KUKA KRL program: EPS_2_251692_SAMH06_A_20251205090702.src

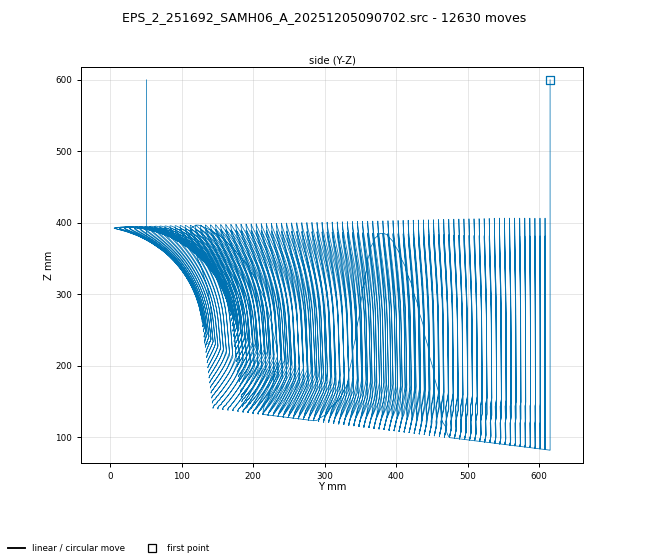
[picture p0: tool path of EPS_2_251692_SAMH06_A_20251205090702.src, 12630 of 12632 moves have a stored position in this frame; points joined in program order, loops and branches not executed]
&ACCESS RVP
&REL 4
&COMMENT QRS 19112012
&PARAM EDITMASK = *
DEF PART()
EXT BAS (BAS_COMMAND :IN,REAL :IN )
INT I
BAS (#INITMOV,0 )

;KUKA QRS Post kuka4.cps  Date:22-06-2017 !

File_ID=2948

QRS_PRE_INIT()

;Init var - Until changes are made in qrs_pre_init
Outlet_Square_prg=0
Inlet_1_Square_prg=0
Inlet_2_Square_prg=0
Inlet_3_Square_prg=0
Inlet_4_Square_prg=0
Inlet_5_Square_prg=0

Outlet_1={X 0.000, Y 543.810, Z 281.000, B 0.000, E1 0.000 }
Inlet_1={X 0.000, Y 545.610, Z 256.000, B 0.000, E1 186.000 }
Outlet_1_type=251
Inlet_1_type=251
;QRS#1=Sidecore dimensions
;QRS#2=250-10" PVC SDR 35
;QRS#3=250-10" PVC SDR 35
;QRS#4=
;QRS#5=
;QRS#6=
;QRS#7=
;QRS#8=
;QRS#9=14M PSX
;QRS#10=14M PSX
;QRS#11=
;QRS#12=
;QRS#13=
;QRS#14=
;QRS#15=
;QRS#16=1220x127x686 2,25'
;QRS#17=EPS Height
;QRS#18=406,5
;QRS#19=*
;QRS#20= UPDATED VERSION 22-06-2017
;QRS#21=*
Outlet_Square=0100
Inlet_1_Square=0100
Inlet_2_Square=0
Inlet_3_Square=0
Inlet_4_Square=0
Inlet_5_Square=0
Mill_Square=1
Outlet_Square_Prg=205
Inlet_1_Square_prg=205

QRS_INIT()

$ADVANCE=5

; T1
PTP {E1 173.621,E2 173.621}
PTP {X 0,Y 615.479,A -85,B 0,C 180,E1 173.621,E2 173.621,E3 0,E4 0,E5 0,E6 0}
QRS_SPEED_INIT()
LIN {X 0,Y 615.479,Z 600,A -85,B 0,C 180,E1 173.621,E2 173.621,E3 0,E4 0,E5 0,E6 0} C_VEL
LIN {X 0,Y 615.479,Z 91.999,A -85,B 0,C 180,E1 173.621,E2 173.621} C_VEL
LIN {X 0,Y 615.479,Z 83.818,A -85,B 0,C 180,E1 173.621,E2 173.621} C_VEL
LIN {X 0,Y 615.469,Z 81.818,A -85,B 0,C 180,E1 173.435,E2 173.435} C_VEL
LIN {X 0,Y 615.495,Z 81.807,A -85,B 0,C 180,E1 170.801,E2 170.801} C_VEL
LIN {X 0,Y 615.489,Z 81.826,A -85,B 0,C 180,E1 168.139,E2 168.139} C_VEL
LIN {X 0,Y 615.464,Z 81.815,A -85,B 0,C 180,E1 165.45,E2 165.45} C_VEL
LIN {X 0,Y 615.485,Z 81.814,A -85,B 0,C 180,E1 162.729,E2 162.729} C_VEL
LIN {X 0,Y 615.469,Z 81.82,A -85,B 0,C 180,E1 159.966,E2 159.966} C_VEL
LIN {X 0,Y 615.486,Z 81.81,A -85,B 0,C 180,E1 157.155,E2 157.155} C_VEL
LIN {X 0,Y 615.476,Z 81.822,A -85,B 0,C 180,E1 154.284,E2 154.284} C_VEL
LIN {X 0,Y 615.47,Z 81.812,A -85,B 0,C 180,E1 151.552,E2 151.552} C_VEL
LIN {X 0,Y 615.492,Z 81.82,A -85,B 0,C 180,E1 148.913,E2 148.913} C_VEL
LIN {X 0,Y 615.47,Z 81.821,A -85,B 0,C 180,E1 146.468,E2 146.468} C_VEL
LIN {X 0,Y 615.458,Z 81.816,A -85,B 0,C 180,E1 144.17,E2 144.17} C_VEL
LIN {X 0,Y 615.467,Z 81.813,A -85,B 0,C 180,E1 141.93,E2 141.93} C_VEL
LIN {X 0,Y 615.492,Z 81.815,A -85,B 0,C 180,E1 139.394,E2 139.394} C_VEL
LIN {X 0,Y 615.466,Z 81.821,A -85,B 0,C 180,E1 136.753,E2 136.753} C_VEL
LIN {X 0,Y 615.474,Z 81.812,A -85,B 0,C 180,E1 133.996,E2 133.996} C_VEL
LIN {X 0,Y 615.475,Z 81.823,A -85,B 0,C 180,E1 131.093,E2 131.093} C_VEL
LIN {X 0,Y 615.459,Z 81.82,A -85,B 0,C 180,E1 128.906,E2 128.906} C_VEL
LIN {X 0,Y 615.46,Z 81.814,A -85,B 0,C 180,E1 126.426,E2 126.426} C_VEL
LIN {X 0,Y 615.494,Z 81.826,A -85,B 0,C 180,E1 123.535,E2 123.535} C_VEL
LIN {X 0,Y 615.45,Z 81.818,A -85,B 0,C 180,E1 120.922,E2 120.922} C_VEL
LIN {X 0,Y 615.474,Z 81.813,A -85,B 0,C 180,E1 118.447,E2 118.447} C_VEL
LIN {X 0,Y 615.471,Z 81.823,A -85,B 0,C 180,E1 115.565,E2 115.565} C_VEL
LIN {X 0,Y 615.465,Z 81.822,A -85,B 0,C 180,E1 113.557,E2 113.557} C_VEL
LIN {X 0,Y 615.453,Z 81.82,A -85,B 0,C 180,E1 111.433,E2 111.433} C_VEL
LIN {X 0,Y 615.447,Z 81.819,A -85,B 0,C 180,E1 109.339,E2 109.339} C_VEL
LIN {X 0,Y 615.485,Z 81.814,A -85,B 0,C 180,E1 106.587,E2 106.587} C_VEL
LIN {X 0,Y 615.468,Z 81.896,A -85,B 0,C 180,E1 104.866,E2 104.866} C_VEL
LIN {X 0,Y 615.446,Z 101.823,A -85,B 0,C 180,E1 102.029,E2 102.029} C_VEL
LIN {X 0,Y 615.452,Z 119.452,A -85,B 0,C 180,E1 99.551,E2 99.551} C_VEL
LIN {X 0,Y 615.46,Z 256.695,A -85,B 0,C 180,E1 97.896,E2 97.896} C_VEL
LIN {X 0,Y 615.48,Z 271.017,A -85,B 0,C 180,E1 97.587,E2 97.587} C_VEL
LIN {X 0,Y 615.491,Z 285.222,A -85,B 0,C 180,E1 97.136,E2 97.136} C_VEL
LIN {X 0,Y 615.494,Z 298.839,A -85,B 0,C 180,E1 96.556,E2 96.556} C_VEL
LIN {X 0,Y 615.49,Z 311.023,A -85,B 0,C 180,E1 95.898,E2 95.898} C_VEL
LIN {X 0,Y 615.498,Z 322.188,A -85,B 0,C 180,E1 95.159,E2 95.159} C_VEL
LIN {X 0,Y 615.497,Z 333.436,A -85,B 0,C 180,E1 94.256,E2 94.256} C_VEL
LIN {X 0,Y 615.496,Z 343.522,A -85,B 0,C 180,E1 93.273,E2 93.273} C_VEL
LIN {X 0,Y 615.497,Z 351.879,A -85,B 0,C 180,E1 92.29,E2 92.29} C_VEL
LIN {X 0,Y 615.496,Z 359.883,A -85,B 0,C 180,E1 91.145,E2 91.145} C_VEL
LIN {X 0,Y 615.494,Z 366.357,A -85,B 0,C 180,E1 90,E2 90} C_VEL
LIN {X 0,Y 615.498,Z 372.115,A -85,B 0,C 180,E1 88.691,E2 88.691} C_VEL
LIN {X 0,Y 615.493,Z 376.34,A -85,B 0,C 180,E1 87.382,E2 87.382} C_VEL
LIN {X 0,Y 615.493,Z 379.15,A -85,B 0,C 180,E1 86.071,E2 86.071} C_VEL
LIN {X 0,Y 615.49,Z 380.617,A -85,B 0,C 180,E1 84.759,E2 84.759} C_VEL
LIN {X 0,Y 615.496,Z 380.768,A -85,B 0,C 180,E1 83.418,E2 83.418} C_VEL
LIN {X 0,Y 615.493,Z 379.611,A -85,B 0,C 180,E1 82.124,E2 82.124} C_VEL
LIN {X 0,Y 615.496,Z 377.073,A -85,B 0,C 180,E1 80.801,E2 80.801} C_VEL
LIN {X 0,Y 615.494,Z 373.067,A -85,B 0,C 180,E1 79.473,E2 79.473} C_VEL
LIN {X 0,Y 615.494,Z 367.474,A -85,B 0,C 180,E1 78.139,E2 78.139} C_VEL
LIN {X 0,Y 615.494,Z 361.111,A -85,B 0,C 180,E1 76.967,E2 76.967} C_VEL
LIN {X 0,Y 615.495,Z 352.912,A -85,B 0,C 180,E1 75.758,E2 75.758} C_VEL
LIN {X 0,Y 615.495,Z 344.746,A -85,B 0,C 180,E1 74.774,E2 74.774} C_VEL
LIN {X 0,Y 615.498,Z 335.393,A -85,B 0,C 180,E1 73.832,E2 73.832} C_VEL
LIN {X 0,Y 615.497,Z 324.257,A -85,B 0,C 180,E1 72.901,E2 72.901} C_VEL
LIN {X 0,Y 615.495,Z 313,A -85,B 0,C 180,E1 72.129,E2 72.129} C_VEL
LIN {X 0,Y 615.497,Z 301.366,A -85,B 0,C 180,E1 71.475,E2 71.475} C_VEL
LIN {X 0,Y 615.483,Z 288.017,A -85,B 0,C 180,E1 70.878,E2 70.878} C_VEL
LIN {X 0,Y 615.495,Z 275.413,A -85,B 0,C 180,E1 70.445,E2 70.445} C_VEL
LIN {X 0,Y 615.477,Z 261.216,A -85,B 0,C 180,E1 70.097,E2 70.097} C_VEL
LIN {X 0,Y 615.478,Z 244.533,A -85,B 0,C 180,E1 69.852,E2 69.852} C_VEL
LIN {X 0,Y 615.468,Z 119.526,A -85,B 0,C 180,E1 68.37,E2 68.37} C_VEL
LIN {X 0,Y 615.494,Z 99.456,A -85,B 0,C 180,E1 65.549,E2 65.549} C_VEL
LIN {X 0,Y 615.42,Z 81.825,A -85,B 0,C 180,E1 63.023,E2 63.023} C_VEL
LIN {X 0,Y 615.417,Z 81.825,A -85,B 0,C 180,E1 60.59,E2 60.59} C_VEL
LIN {X 0,Y 615.445,Z 81.825,A -85,B 0,C 180,E1 58.312,E2 58.312} C_VEL
LIN {X 0,Y 615.494,Z 81.826,A -85,B 0,C 180,E1 55.978,E2 55.978} C_VEL
LIN {X 0,Y 615.443,Z 81.823,A -85,B 0,C 180,E1 53.572,E2 53.572} C_VEL
LIN {X 0,Y 615.424,Z 81.824,A -85,B 0,C 180,E1 50.946,E2 50.946} C_VEL
LIN {X 0,Y 615.464,Z 81.825,A -85,B 0,C 180,E1 48.524,E2 48.524} C_VEL
LIN {X 0,Y 615.449,Z 81.822,A -85,B 0,C 180,E1 45.847,E2 45.847} C_VEL
LIN {X 0,Y 615.428,Z 81.823,A -85,B 0,C 180,E1 43.25,E2 43.25} C_VEL
LIN {X 0,Y 615.487,Z 81.826,A -85,B 0,C 180,E1 40.607,E2 40.607} C_VEL
LIN {X 0,Y 615.449,Z 81.819,A -85,B 0,C 180,E1 38.007,E2 38.007} C_VEL
LIN {X 0,Y 615.432,Z 81.821,A -85,B 0,C 180,E1 35.62,E2 35.62} C_VEL
LIN {X 0,Y 615.453,Z 81.823,A -85,B 0,C 180,E1 33.239,E2 33.239} C_VEL
LIN {X 0,Y 615.49,Z 81.827,A -85,B 0,C 180,E1 30.92,E2 30.92} C_VEL
LIN {X 0,Y 615.437,Z 81.82,A -85,B 0,C 180,E1 27.918,E2 27.918} C_VEL
LIN {X 0,Y 615.452,Z 81.822,A -85,B 0,C 180,E1 25.562,E2 25.562} C_VEL
LIN {X 0,Y 615.486,Z 81.816,A -85,B 0,C 180,E1 22.845,E2 22.845} C_VEL
LIN {X 0,Y 615.443,Z 81.82,A -85,B 0,C 180,E1 20.034,E2 20.034} C_VEL
LIN {X 0,Y 615.496,Z 81.821,A -85,B 0,C 180,E1 17.27,E2 17.27} C_VEL
LIN {X 0,Y 615.448,Z 81.817,A -85,B 0,C 180,E1 14.55,E2 14.55} C_VEL
LIN {X 0,Y 615.449,Z 81.817,A -85,B 0,C 180,E1 12.531,E2 12.531} C_VEL
LIN {X 0,Y 615.48,Z 81.824,A -85,B 0,C 180,E1 9.862,E2 9.862} C_VEL
LIN {X 0,Y 615.481,Z 81.813,A -85,B 0,C 180,E1 7.216,E2 7.216} C_VEL
LIN {X 0,Y 615.452,Z 81.818,A -85,B 0,C 180,E1 4.585,E2 4.585} C_VEL
LIN {X 0,Y 615.498,Z 81.825,A -85,B 0,C 180,E1 1.963,E2 1.963} C_VEL
LIN {X 0,Y 615.476,Z 81.812,A -85,B 0,C 180,E1 -0.654,E2 -0.654} C_VEL
LIN {X 0,Y 615.459,Z 81.819,A -85,B 0,C 180,E1 -3.273,E2 -3.273} C_VEL
LIN {X 0,Y 615.493,Z 81.82,A -85,B 0,C 180,E1 -5.898,E2 -5.898} C_VEL
LIN {X 0,Y 615.474,Z 81.811,A -85,B 0,C 180,E1 -8.537,E2 -8.537} C_VEL
LIN {X 0,Y 615.47,Z 81.821,A -85,B 0,C 180,E1 -11.193,E2 -11.193} C_VEL
LIN {X 0,Y 615.49,Z 81.813,A -85,B 0,C 180,E1 -13.933,E2 -13.933} C_VEL
LIN {X 0,Y 615.462,Z 81.815,A -85,B 0,C 180,E1 -16.587,E2 -16.587} C_VEL
LIN {X 0,Y 615.493,Z 81.823,A -85,B 0,C 180,E1 -19.338,E2 -19.338} C_VEL
LIN {X 0,Y 615.469,Z 81.813,A -85,B 0,C 180,E1 -22.342,E2 -22.342} C_VEL
LIN {X 0,Y 615.492,Z 81.826,A -85,B 0,C 180,E1 -24.992,E2 -24.992} C_VEL
LIN {X 0,Y 615.484,Z 81.809,A -85,B 0,C 180,E1 -27.915,E2 -27.915} C_VEL
LIN {X 0,Y 615.471,Z 81.814,A -85,B 0,C 180,E1 -30.161,E2 -30.161} C_VEL
LIN {X 0,Y 615.478,Z 81.82,A -85,B 0,C 180,E1 -32.458,E2 -32.458} C_VEL
LIN {X 0,Y 615.49,Z 81.822,A -85,B 0,C 180,E1 -34.815,E2 -34.815} C_VEL
LIN {X 0,Y 615.487,Z 81.81,A -85,B 0,C 180,E1 -37.242,E2 -37.242} C_VEL
LIN {X 0,Y 615.476,Z 81.818,A -85,B 0,C 180,E1 -40.088,E2 -40.088} C_VEL
LIN {X 0,Y 615.497,Z 81.825,A -85,B 0,C 180,E1 -42.352,E2 -42.352} C_VEL
LIN {X 0,Y 615.481,Z 81.811,A -85,B 0,C 180,E1 -45.069,E2 -45.069} C_VEL
LIN {X 0,Y 615.483,Z 81.82,A -85,B 0,C 180,E1 -47.92,E2 -47.92} C_VEL
LIN {X 0,Y 615.486,Z 81.823,A -85,B 0,C 180,E1 -50.25,E2 -50.25} C_VEL
LIN {X 0,Y 615.489,Z 81.808,A -85,B 0,C 180,E1 -53.063,E2 -53.063} C_VEL
LIN {X 0,Y 615.492,Z 81.823,A -85,B 0,C 180,E1 -55.978,E2 -55.978} C_VEL
LIN {X 0,Y 615.488,Z 81.809,A -85,B 0,C 180,E1 -58.914,E2 -58.914} C_VEL
LIN {X 0,Y 615.492,Z 81.822,A -85,B 0,C 180,E1 -61.549,E2 -61.549} C_VEL
LIN {X 0,Y 615.479,Z 81.81,A -85,B 0,C 180,E1 -64.433,E2 -64.433} C_VEL
LIN {X 0,Y 615.492,Z 81.815,A -85,B 0,C 180,E1 -66.711,E2 -66.711} C_VEL
LIN {X 0,Y 615.483,Z 104.503,A -85,B 0,C 180,E1 -69.576,E2 -69.576} C_VEL
LIN {X 0,Y 615.496,Z 127.142,A -85,B 0,C 180,E1 -72.387,E2 -72.387} C_VEL
LIN {X 0,Y 615.494,Z 143.505,A -85,B 0,C 180,E1 -74.392,E2 -74.392} C_VEL
LIN {X 0,Y 615.478,Z 281.308,A -85,B 0,C 180,E1 -76.052,E2 -76.052} C_VEL
LIN {X 0,Y 615.489,Z 294.854,A -85,B 0,C 180,E1 -76.336,E2 -76.336} C_VEL
LIN {X 0,Y 615.488,Z 308.565,A -85,B 0,C 180,E1 -76.757,E2 -76.757} C_VEL
LIN {X 0,Y 615.494,Z 321.835,A -85,B 0,C 180,E1 -77.302,E2 -77.302} C_VEL
LIN {X 0,Y 615.483,Z 334.599,A -85,B 0,C 180,E1 -77.972,E2 -77.972} C_VEL
LIN {X 0,Y 615.499,Z 347.339,A -85,B 0,C 180,E1 -78.807,E2 -78.807} C_VEL
LIN {X 0,Y 615.498,Z 357.747,A -85,B 0,C 180,E1 -79.639,E2 -79.639} C_VEL
LIN {X 0,Y 615.496,Z 368.087,A -85,B 0,C 180,E1 -80.636,E2 -80.636} C_VEL
LIN {X 0,Y 615.497,Z 376.602,A -85,B 0,C 180,E1 -81.629,E2 -81.629} C_VEL
LIN {X 0,Y 615.496,Z 384.726,A -85,B 0,C 180,E1 -82.784,E2 -82.784} C_VEL
LIN {X 0,Y 615.496,Z 390.429,A -85,B 0,C 180,E1 -83.772,E2 -83.772} C_VEL
LIN {X 0,Y 615.495,Z 395.08,A -85,B 0,C 180,E1 -84.759,E2 -84.759} C_VEL
LIN {X 0,Y 615.496,Z 399.901,A -85,B 0,C 180,E1 -86.071,E2 -86.071} C_VEL
LIN {X 0,Y 615.495,Z 403.252,A -85,B 0,C 180,E1 -87.382,E2 -87.382} C_VEL
LIN {X 0,Y 615.49,Z 405.228,A -85,B 0,C 180,E1 -88.691,E2 -88.691} C_VEL
LIN {X 0,Y 615.493,Z 405.889,A -85,B 0,C 180,E1 -90,E2 -90} C_VEL
LIN {X 0,Y 615.49,Z 405.229,A -85,B 0,C 180,E1 -91.308,E2 -91.308} C_VEL
LIN {X 0,Y 615.495,Z 403.252,A -85,B 0,C 180,E1 -92.618,E2 -92.618} C_VEL
LIN {X 0,Y 615.496,Z 399.901,A -85,B 0,C 180,E1 -93.928,E2 -93.928} C_VEL
LIN {X 0,Y 615.495,Z 395.081,A -85,B 0,C 180,E1 -95.241,E2 -95.241} C_VEL
LIN {X 0,Y 615.495,Z 388.629,A -85,B 0,C 180,E1 -96.556,E2 -96.556} C_VEL
LIN {X 0,Y 615.498,Z 381.441,A -85,B 0,C 180,E1 -97.71,E2 -97.71} C_VEL
LIN {X 0,Y 615.497,Z 373.904,A -85,B 0,C 180,E1 -98.702,E2 -98.702} C_VEL
LIN {X 0,Y 615.496,Z 364.854,A -85,B 0,C 180,E1 -99.696,E2 -99.696} C_VEL
LIN {X 0,Y 615.497,Z 354.758,A -85,B 0,C 180,E1 -100.618,E2 -100.618} C_VEL
LIN {X 0,Y 615.498,Z 343.859,A -85,B 0,C 180,E1 -101.443,E2 -101.443} C_VEL
LIN {X 0,Y 615.484,Z 331.708,A -85,B 0,C 180,E1 -102.195,E2 -102.195} C_VEL
LIN {X 0,Y 615.486,Z 318.093,A -85,B 0,C 180,E1 -102.865,E2 -102.865} C_VEL
LIN {X 0,Y 615.488,Z 304.838,A -85,B 0,C 180,E1 -103.369,E2 -103.369} C_VEL
LIN {X 0,Y 615.487,Z 291.29,A -85,B 0,C 180,E1 -103.748,E2 -103.748} C_VEL
LIN {X 0,Y 615.479,Z 277.161,A -85,B 0,C 180,E1 -104.007,E2 -104.007} C_VEL
LIN {X 0,Y 615.494,Z 143.507,A -85,B 0,C 180,E1 -105.607,E2 -105.607} C_VEL
LIN {X 0,Y 615.471,Z 120.463,A -85,B 0,C 180,E1 -108.439,E2 -108.439} C_VEL
LIN {X 0,Y 615.472,Z 99.26,A -85,B 0,C 180,E1 -111.081,E2 -111.081} C_VEL
LIN {X 0,Y 615.494,Z 81.808,A -85,B 0,C 180,E1 -113.311,E2 -113.311} C_VEL
LIN {X 0,Y 615.473,Z 81.813,A -85,B 0,C 180,E1 -115.716,E2 -115.716} C_VEL
LIN {X 0,Y 615.493,Z 81.823,A -85,B 0,C 180,E1 -118.451,E2 -118.451} C_VEL
LIN {X 0,Y 615.486,Z 81.809,A -85,B 0,C 180,E1 -121.086,E2 -121.086} C_VEL
LIN {X 0,Y 615.474,Z 81.814,A -85,B 0,C 180,E1 -123.532,E2 -123.532} C_VEL
LIN {X 0,Y 615.481,Z 81.82,A -85,B 0,C 180,E1 -125.833,E2 -125.833} C_VEL
LIN {X 0,Y 615.488,Z 81.826,A -85,B 0,C 180,E1 -128.068,E2 -128.068} C_VEL
LIN {X 0,Y 615.479,Z 81.812,A -85,B 0,C 180,E1 -130.607,E2 -130.607} C_VEL
LIN {X 0,Y 615.474,Z 81.814,A -85,B 0,C 180,E1 -133.246,E2 -133.246} C_VEL
LIN {X 0,Y 615.485,Z 81.82,A -85,B 0,C 180,E1 -136.003,E2 -136.003} C_VEL
LIN {X 0,Y 615.487,Z 81.809,A -85,B 0,C 180,E1 -138.526,E2 -138.526} C_VEL
LIN {X 0,Y 615.477,Z 81.815,A -85,B 0,C 180,E1 -141.095,E2 -141.095} C_VEL
LIN {X 0,Y 615.483,Z 81.827,A -85,B 0,C 180,E1 -143.575,E2 -143.575} C_VEL
LIN {X 0,Y 615.494,Z 81.807,A -85,B 0,C 180,E1 -146.464,E2 -146.464} C_VEL
LIN {X 0,Y 615.484,Z 81.82,A -85,B 0,C 180,E1 -149.08,E2 -149.08} C_VEL
LIN {X 0,Y 615.477,Z 81.82,A -85,B 0,C 180,E1 -151.551,E2 -151.551} C_VEL
LIN {X 0,Y 615.486,Z 81.81,A -85,B 0,C 180,E1 -154.431,E2 -154.431} C_VEL
LIN {X 0,Y 615.485,Z 81.825,A -85,B 0,C 180,E1 -157.155,E2 -157.155} C_VEL
LIN {X 0,Y 615.485,Z 81.809,A -85,B 0,C 180,E1 -159.967,E2 -159.967} C_VEL
LIN {X 0,Y 615.488,Z 81.822,A -85,B 0,C 180,E1 -162.73,E2 -162.73} C_VEL
LIN {X 0,Y 615.474,Z 81.813,A -85,B 0,C 180,E1 -165.451,E2 -165.451} C_VEL
LIN {X 0,Y 615.485,Z 81.813,A -85,B 0,C 180,E1 -168.139,E2 -168.139} C_VEL
LIN {X 0,Y 615.484,Z 81.822,A -85,B 0,C 180,E1 -170.801,E2 -170.801} C_VEL
LIN {X 0,Y 615.481,Z 81.81,A -85,B 0,C 180,E1 -173.443,E2 -173.443} C_VEL
LIN {X 0,Y 615.485,Z 81.817,A -85,B 0,C 180,E1 -176.072,E2 -176.072} C_VEL
LIN {X 0,Y 615.475,Z 81.82,A -85,B 0,C 180,E1 -178.691,E2 -178.691} C_VEL
LIN {X 0,Y 615.486,Z 81.808,A -85,B 0,C 180,E1 -181.309,E2 -181.309} C_VEL
LIN {X 0,Y 615.488,Z 81.819,A -85,B 0,C 180,E1 -183.929,E2 -183.929} C_VEL
LIN {X 0,Y 615.469,Z 81.818,A -85,B 0,C 180,E1 -186.565,E2 -186.565} C_VEL
LIN {X 0,Y 614.805,Z 81.958,A -85,B 0,C 180,E1 -187.111,E2 -187.111} C_VEL
LIN {X 0,Y 611.984,Z 82.383,A -85,B 0,C 180,E1 -187.997,E2 -187.997} C_VEL
LIN {X 0,Y 609.596,Z 82.686,A -85,B 0,C 180,E1 -188.71,E2 -188.71} C_VEL
LIN {X 0,Y 608.558,Z 82.802,A -85,B 0,C 180,E1 -189.259,E2 -189.259} C_VEL
LIN {X 0,Y 608.467,Z 82.813,A -85,B 0,C 180,E1 -189.445,E2 -189.445} C_VEL
LIN {X 0,Y 608.46,Z 82.821,A -85,B 0,C 180,E1 -192,E2 -192} C_VEL
LIN {X 0,Y 608.463,Z 82.812,A -85,B 0,C 180,E1 -194.721,E2 -194.721} C_VEL
LIN {X 0,Y 608.45,Z 82.819,A -85,B 0,C 180,E1 -197.477,E2 -197.477} C_VEL
LIN {X 0,Y 608.447,Z 82.815,A -85,B 0,C 180,E1 -200.275,E2 -200.275} C_VEL
LIN {X 0,Y 608.458,Z 82.812,A -85,B 0,C 180,E1 -202.477,E2 -202.477} C_VEL
LIN {X 0,Y 608.454,Z 82.82,A -85,B 0,C 180,E1 -205.301,E2 -205.301} C_VEL
LIN {X 0,Y 608.442,Z 82.822,A -85,B 0,C 180,E1 -207.519,E2 -207.519} C_VEL
LIN {X 0,Y 608.445,Z 82.815,A -85,B 0,C 180,E1 -209.968,E2 -209.968} C_VEL
LIN {X 0,Y 608.455,Z 82.817,A -85,B 0,C 180,E1 -212.88,E2 -212.88} C_VEL
LIN {X 0,Y 608.432,Z 82.823,A -85,B 0,C 180,E1 -215.279,E2 -215.279} C_VEL
LIN {X 0,Y 608.455,Z 82.813,A -85,B 0,C 180,E1 -217.748,E2 -217.748} C_VEL
LIN {X 0,Y 608.445,Z 82.815,A -85,B 0,C 180,E1 -220.329,E2 -220.329} C_VEL
LIN {X 0,Y 608.451,Z 82.822,A -85,B 0,C 180,E1 -222.96,E2 -222.96} C_VEL
LIN {X 0,Y 608.436,Z 82.815,A -85,B 0,C 180,E1 -225.738,E2 -225.738} C_VEL
LIN {X 0,Y 608.454,Z 82.813,A -85,B 0,C 180,E1 -227.938,E2 -227.938} C_VEL
LIN {X 0,Y 608.439,Z 82.824,A -85,B 0,C 180,E1 -230.707,E2 -230.707} C_VEL
LIN {X 0,Y 608.428,Z 82.818,A -85,B 0,C 180,E1 -233.083,E2 -233.083} C_VEL
LIN {X 0,Y 608.452,Z 82.813,A -85,B 0,C 180,E1 -235.53,E2 -235.53} C_VEL
LIN {X 0,Y 608.462,Z 82.814,A -85,B 0,C 180,E1 -237.906,E2 -237.906} C_VEL
LIN {X 0,Y 608.479,Z 82.818,A -85,B 0,C 180,E1 -240.221,E2 -240.221} C_VEL
LIN {X 0,Y 608.429,Z 82.818,A -85,B 0,C 180,E1 -242.803,E2 -242.803} C_VEL
LIN {X 0,Y 608.443,Z 82.815,A -85,B 0,C 180,E1 -245.429,E2 -245.429} C_VEL
LIN {X 0,Y 608.453,Z 82.819,A -85,B 0,C 180,E1 -248.308,E2 -248.308} C_VEL
LIN {X 0,Y 608.447,Z 82.814,A -85,B 0,C 180,E1 -251.13,E2 -251.13} C_VEL
LIN {X 0,Y 608.454,Z 82.823,A -85,B 0,C 180,E1 -253.906,E2 -253.906} C_VEL
LIN {X 0,Y 608.443,Z 82.879,A -85,B 0,C 180,E1 -255.022,E2 -255.022} C_VEL
LIN {X 0,Y 608.505,Z 100.007,A -85,B 0,C 180,E1 -257.493,E2 -257.493} C_VEL
LIN {X 0,Y 608.468,Z 119.013,A -85,B 0,C 180,E1 -260.191,E2 -260.191} C_VEL
LIN {X 0,Y 608.509,Z 119.95,A -85,B 0,C 180,E1 -260.286,E2 -260.286} C_VEL
LIN {X 0,Y 608.592,Z 255.971,A -85,B 0,C 180,E1 -261.93,E2 -261.93} C_VEL
LIN {X 0,Y 608.571,Z 270.582,A -85,B 0,C 180,E1 -262.243,E2 -262.243} C_VEL
LIN {X 0,Y 608.587,Z 283.896,A -85,B 0,C 180,E1 -262.661,E2 -262.661} C_VEL
LIN {X 0,Y 608.544,Z 297.268,A -85,B 0,C 180,E1 -263.219,E2 -263.219} C_VEL
LIN {X 0,Y 608.526,Z 309.517,A -85,B 0,C 180,E1 -263.867,E2 -263.867} C_VEL
LIN {X 0,Y 608.502,Z 322.152,A -85,B 0,C 180,E1 -264.699,E2 -264.699} C_VEL
LIN {X 0,Y 608.49,Z 332.525,A -85,B 0,C 180,E1 -265.529,E2 -265.529} C_VEL
LIN {X 0,Y 608.472,Z 342.87,A -85,B 0,C 180,E1 -266.524,E2 -266.524} C_VEL
LIN {X 0,Y 608.464,Z 351.439,A -85,B 0,C 180,E1 -267.518,E2 -267.518} C_VEL
LIN {X 0,Y 608.45,Z 359.687,A -85,B 0,C 180,E1 -268.676,E2 -268.676} C_VEL
LIN {X 0,Y 608.441,Z 365.452,A -85,B 0,C 180,E1 -269.669,E2 -269.669} C_VEL
LIN {X 0,Y 608.448,Z 371.636,A -85,B 0,C 180,E1 -270.993,E2 -270.993} C_VEL
LIN {X 0,Y 608.441,Z 375.17,A -85,B 0,C 180,E1 -271.986,E2 -271.986} C_VEL
LIN {X 0,Y 608.418,Z 378.646,A -85,B 0,C 180,E1 -273.311,E2 -273.311} C_VEL
LIN {X 0,Y 608.429,Z 380.732,A -85,B 0,C 180,E1 -274.638,E2 -274.638} C_VEL
LIN {X 0,Y 608.431,Z 381.488,A -85,B 0,C 180,E1 -275.967,E2 -275.967} C_VEL
LIN {X 0,Y 608.42,Z 380.907,A -85,B 0,C 180,E1 -277.3,E2 -277.3} C_VEL
LIN {X 0,Y 608.42,Z 378.953,A -85,B 0,C 180,E1 -278.637,E2 -278.637} C_VEL
LIN {X 0,Y 608.434,Z 375.573,A -85,B 0,C 180,E1 -279.978,E2 -279.978} C_VEL
LIN {X 0,Y 608.429,Z 370.663,A -85,B 0,C 180,E1 -281.325,E2 -281.325} C_VEL
LIN {X 0,Y 608.457,Z 365.899,A -85,B 0,C 180,E1 -282.338,E2 -282.338} C_VEL
LIN {X 0,Y 608.459,Z 358.935,A -85,B 0,C 180,E1 -283.527,E2 -283.527} C_VEL
LIN {X 0,Y 608.457,Z 351.621,A -85,B 0,C 180,E1 -284.55,E2 -284.55} C_VEL
LIN {X 0,Y 608.471,Z 342.76,A -85,B 0,C 180,E1 -285.578,E2 -285.578} C_VEL
LIN {X 0,Y 608.495,Z 332.04,A -85,B 0,C 180,E1 -286.603,E2 -286.603} C_VEL
LIN {X 0,Y 608.511,Z 321.001,A -85,B 0,C 180,E1 -287.475,E2 -287.475} C_VEL
LIN {X 0,Y 608.524,Z 309.03,A -85,B 0,C 180,E1 -288.252,E2 -288.252} C_VEL
LIN {X 0,Y 608.543,Z 297.362,A -85,B 0,C 180,E1 -288.867,E2 -288.867} C_VEL
LIN {X 0,Y 608.577,Z 283.761,A -85,B 0,C 180,E1 -289.435,E2 -289.435} C_VEL
LIN {X 0,Y 608.58,Z 269.596,A -85,B 0,C 180,E1 -289.874,E2 -289.874} C_VEL
LIN {X 0,Y 608.608,Z 255.992,A -85,B 0,C 180,E1 -290.159,E2 -290.159} C_VEL
LIN {X 0,Y 608.555,Z 120.203,A -85,B 0,C 180,E1 -291.8,E2 -291.8} C_VEL
LIN {X 0,Y 608.471,Z 119.536,A -85,B 0,C 180,E1 -291.825,E2 -291.825} C_VEL
LIN {X 0,Y 608.52,Z 100.202,A -85,B 0,C 180,E1 -294.568,E2 -294.568} C_VEL
LIN {X 0,Y 608.494,Z 83.884,A -85,B 0,C 180,E1 -296.92,E2 -296.92} C_VEL
LIN {X 0,Y 608.4,Z 82.821,A -85,B 0,C 180,E1 -297.12,E2 -297.12} C_VEL
LIN {X 0,Y 608.448,Z 82.821,A -85,B 0,C 180,E1 -299.968,E2 -299.968} C_VEL
LIN {X 0,Y 608.413,Z 82.818,A -85,B 0,C 180,E1 -302.882,E2 -302.882} C_VEL
LIN {X 0,Y 608.404,Z 82.82,A -85,B 0,C 180,E1 -305.28,E2 -305.28} C_VEL
LIN {X 0,Y 608.422,Z 82.821,A -85,B 0,C 180,E1 -308.234,E2 -308.234} C_VEL
LIN {X 0,Y 608.435,Z 82.817,A -85,B 0,C 180,E1 -310.327,E2 -310.327} C_VEL
LIN {X 0,Y 608.398,Z 82.821,A -85,B 0,C 180,E1 -312.965,E2 -312.965} C_VEL
LIN {X 0,Y 608.448,Z 82.821,A -85,B 0,C 180,E1 -315.737,E2 -315.737} C_VEL
LIN {X 0,Y 608.445,Z 82.817,A -85,B 0,C 180,E1 -317.937,E2 -317.937} C_VEL
LIN {X 0,Y 608.413,Z 82.819,A -85,B 0,C 180,E1 -320.709,E2 -320.709} C_VEL
LIN {X 0,Y 608.434,Z 82.822,A -85,B 0,C 180,E1 -323.083,E2 -323.083} C_VEL
LIN {X 0,Y 608.465,Z 82.816,A -85,B 0,C 180,E1 -325.53,E2 -325.53} C_VEL
LIN {X 0,Y 608.439,Z 82.815,A -85,B 0,C 180,E1 -327.904,E2 -327.904} C_VEL
LIN {X 0,Y 608.421,Z 82.817,A -85,B 0,C 180,E1 -330.218,E2 -330.218} C_VEL
LIN {X 0,Y 608.46,Z 82.82,A -85,B 0,C 180,E1 -332.796,E2 -332.796} C_VEL
LIN {X 0,Y 608.439,Z 82.816,A -85,B 0,C 180,E1 -335.428,E2 -335.428} C_VEL
LIN {X 0,Y 608.448,Z 82.817,A -85,B 0,C 180,E1 -338.307,E2 -338.307} C_VEL
LIN {X 0,Y 608.456,Z 82.813,A -85,B 0,C 180,E1 -341.288,E2 -341.288} C_VEL
LIN {X 0,Y 608.43,Z 82.817,A -85,B 0,C 180,E1 -343.905,E2 -343.905} C_VEL
LIN {X 0,Y 608.464,Z 82.818,A -85,B 0,C 180,E1 -346.643,E2 -346.643} C_VEL
LIN {X 0,Y 608.435,Z 82.815,A -85,B 0,C 180,E1 -349.35,E2 -349.35} C_VEL
LIN {X 0,Y 608.47,Z 82.817,A -85,B 0,C 180,E1 -352.033,E2 -352.033} C_VEL
LIN {X 0,Y 608.467,Z 82.813,A -85,B 0,C 180,E1 -354.698,E2 -354.698} C_VEL
LIN {X 0,Y 608.447,Z 82.814,A -85,B 0,C 180,E1 -357.352,E2 -357.352} C_VEL
LIN {X 0,Y 608.479,Z 82.819,A -85,B 0,C 180,E1 -360,E2 -360} C_VEL
LIN {X 0,Y 608.47,Z 82.811,A -85,B 0,C 180,E1 -362.648,E2 -362.648} C_VEL
LIN {X 0,Y 608.444,Z 82.817,A -85,B 0,C 180,E1 -365.302,E2 -365.302} C_VEL
LIN {X 0,Y 608.479,Z 82.814,A -85,B 0,C 180,E1 -367.967,E2 -367.967} C_VEL
LIN {X 0,Y 608.453,Z 82.814,A -85,B 0,C 180,E1 -370.948,E2 -370.948} C_VEL
LIN {X 0,Y 608.458,Z 82.821,A -85,B 0,C 180,E1 -373.356,E2 -373.356} C_VEL
LIN {X 0,Y 608.458,Z 82.813,A -85,B 0,C 180,E1 -376.094,E2 -376.094} C_VEL
LIN {X 0,Y 608.449,Z 82.817,A -85,B 0,C 180,E1 -378.87,E2 -378.87} C_VEL
LIN {X 0,Y 608.465,Z 82.813,A -85,B 0,C 180,E1 -381.692,E2 -381.692} C_VEL
LIN {X 0,Y 608.447,Z 82.816,A -85,B 0,C 180,E1 -384.571,E2 -384.571} C_VEL
LIN {X 0,Y 608.479,Z 82.815,A -85,B 0,C 180,E1 -387.207,E2 -387.207} C_VEL
LIN {X 0,Y 608.463,Z 82.812,A -85,B 0,C 180,E1 -389.971,E2 -389.971} C_VEL
LIN {X 0,Y 608.455,Z 82.819,A -85,B 0,C 180,E1 -392.521,E2 -392.521} C_VEL
LIN {X 0,Y 608.448,Z 82.815,A -85,B 0,C 180,E1 -395.277,E2 -395.277} C_VEL
LIN {X 0,Y 608.461,Z 82.812,A -85,B 0,C 180,E1 -397.747,E2 -397.747} C_VEL
LIN {X 0,Y 608.448,Z 82.821,A -85,B 0,C 180,E1 -400.329,E2 -400.329} C_VEL
LIN {X 0,Y 608.481,Z 82.809,A -85,B 0,C 180,E1 -403.31,E2 -403.31} C_VEL
LIN {X 0,Y 608.468,Z 82.819,A -85,B 0,C 180,E1 -406.13,E2 -406.13} C_VEL
LIN {X 0,Y 608.453,Z 82.814,A -85,B 0,C 180,E1 -408.823,E2 -408.823} C_VEL
LIN {X 0,Y 608.473,Z 82.812,A -85,B 0,C 180,E1 -411.412,E2 -411.412} C_VEL
LIN {X 0,Y 608.447,Z 82.824,A -85,B 0,C 180,E1 -413.955,E2 -413.955} C_VEL
LIN {X 0,Y 608.447,Z 82.816,A -85,B 0,C 180,E1 -416.328,E2 -416.328} C_VEL
LIN {X 0,Y 608.449,Z 82.813,A -85,B 0,C 180,E1 -418.732,E2 -418.732} C_VEL
LIN {X 0,Y 608.475,Z 82.815,A -85,B 0,C 180,E1 -421.38,E2 -421.38} C_VEL
LIN {X 0,Y 608.443,Z 82.818,A -85,B 0,C 180,E1 -423.964,E2 -423.964} C_VEL
LIN {X 0,Y 608.492,Z 82.862,A -85,B 0,C 180,E1 -426.562,E2 -426.562} C_VEL
LIN {X 0,Y 608.566,Z 99.259,A -85,B 0,C 180,E1 -428.668,E2 -428.668} C_VEL
LIN {X 0,Y 608.534,Z 119.865,A -85,B 0,C 180,E1 -431.267,E2 -431.267} C_VEL
LIN {X 0,Y 608.523,Z 142.519,A -85,B 0,C 180,E1 -434.08,E2 -434.08} C_VEL
LIN {X 0,Y 608.572,Z 144.031,A -85,B 0,C 180,E1 -434.232,E2 -434.232} C_VEL
LIN {X 0,Y 608.599,Z 281.447,A -85,B 0,C 180,E1 -435.894,E2 -435.894} C_VEL
LIN {X 0,Y 608.604,Z 295.621,A -85,B 0,C 180,E1 -436.2,E2 -436.2} C_VEL
LIN {X 0,Y 608.579,Z 309.708,A -85,B 0,C 180,E1 -436.646,E2 -436.646} C_VEL
LIN {X 0,Y 608.555,Z 321.881,A -85,B 0,C 180,E1 -437.155,E2 -437.155} C_VEL
LIN {X 0,Y 608.511,Z 334.679,A -85,B 0,C 180,E1 -437.832,E2 -437.832} C_VEL
LIN {X 0,Y 608.499,Z 347.469,A -85,B 0,C 180,E1 -438.677,E2 -438.677} C_VEL
LIN {X 0,Y 608.496,Z 357.93,A -85,B 0,C 180,E1 -439.519,E2 -439.519} C_VEL
LIN {X 0,Y 608.479,Z 368.333,A -85,B 0,C 180,E1 -440.527,E2 -440.527} C_VEL
LIN {X 0,Y 608.464,Z 376.913,A -85,B 0,C 180,E1 -441.531,E2 -441.531} C_VEL
LIN {X 0,Y 608.461,Z 385.113,A -85,B 0,C 180,E1 -442.7,E2 -442.7} C_VEL
LIN {X 0,Y 608.444,Z 391.545,A -85,B 0,C 180,E1 -443.831,E2 -443.831} C_VEL
LIN {X 0,Y 608.435,Z 396.961,A -85,B 0,C 180,E1 -445.03,E2 -445.03} C_VEL
LIN {X 0,Y 608.434,Z 400.441,A -85,B 0,C 180,E1 -446.026,E2 -446.026} C_VEL
LIN {X 0,Y 608.423,Z 403.831,A -85,B 0,C 180,E1 -447.352,E2 -447.352} C_VEL
LIN {X 0,Y 608.442,Z 405.83,A -85,B 0,C 180,E1 -448.676,E2 -448.676} C_VEL
LIN {X 0,Y 608.433,Z 406.5,A -85,B 0,C 180,E1 -450,E2 -450} C_VEL
LIN {X 0,Y 608.442,Z 405.831,A -85,B 0,C 180,E1 -451.324,E2 -451.324} C_VEL
LIN {X 0,Y 608.423,Z 403.831,A -85,B 0,C 180,E1 -452.648,E2 -452.648} C_VEL
LIN {X 0,Y 608.434,Z 400.442,A -85,B 0,C 180,E1 -453.974,E2 -453.974} C_VEL
LIN {X 0,Y 608.439,Z 395.568,A -85,B 0,C 180,E1 -455.302,E2 -455.302} C_VEL
LIN {X 0,Y 608.445,Z 389.212,A -85,B 0,C 180,E1 -456.603,E2 -456.603} C_VEL
LIN {X 0,Y 608.454,Z 381.798,A -85,B 0,C 180,E1 -457.8,E2 -457.8} C_VEL
LIN {X 0,Y 608.472,Z 372.824,A -85,B 0,C 180,E1 -458.97,E2 -458.97} C_VEL
LIN {X 0,Y 608.472,Z 363.392,A -85,B 0,C 180,E1 -459.977,E2 -459.977} C_VEL
LIN {X 0,Y 608.505,Z 352.048,A -85,B 0,C 180,E1 -460.973,E2 -460.973} C_VEL
LIN {X 0,Y 608.53,Z 340.15,A -85,B 0,C 180,E1 -461.829,E2 -461.829} C_VEL
LIN {X 0,Y 608.53,Z 327.074,A -85,B 0,C 180,E1 -462.591,E2 -462.591} C_VEL
LIN {X 0,Y 608.55,Z 314.174,A -85,B 0,C 180,E1 -463.184,E2 -463.184} C_VEL
LIN {X 0,Y 608.59,Z 300.184,A -85,B 0,C 180,E1 -463.672,E2 -463.672} C_VEL
LIN {X 0,Y 608.598,Z 286.457,A -85,B 0,C 180,E1 -464.013,E2 -464.013} C_VEL
LIN {X 0,Y 608.619,Z 270.171,A -85,B 0,C 180,E1 -464.257,E2 -464.257} C_VEL
LIN {X 0,Y 608.529,Z 143.655,A -85,B 0,C 180,E1 -465.78,E2 -465.78} C_VEL
LIN {X 0,Y 608.536,Z 121.779,A -85,B 0,C 180,E1 -468.494,E2 -468.494} C_VEL
LIN {X 0,Y 608.556,Z 100.656,A -85,B 0,C 180,E1 -471.155,E2 -471.155} C_VEL
LIN {X 0,Y 608.558,Z 83.212,A -85,B 0,C 180,E1 -473.39,E2 -473.39} C_VEL
LIN {X 0,Y 608.477,Z 82.812,A -85,B 0,C 180,E1 -473.483,E2 -473.483} C_VEL
LIN {X 0,Y 608.442,Z 82.818,A -85,B 0,C 180,E1 -476.036,E2 -476.036} C_VEL
LIN {X 0,Y 608.476,Z 82.816,A -85,B 0,C 180,E1 -478.62,E2 -478.62} C_VEL
LIN {X 0,Y 608.445,Z 82.814,A -85,B 0,C 180,E1 -481.318,E2 -481.318} C_VEL
LIN {X 0,Y 608.472,Z 82.814,A -85,B 0,C 180,E1 -483.735,E2 -483.735} C_VEL
LIN {X 0,Y 608.446,Z 82.824,A -85,B 0,C 180,E1 -486.092,E2 -486.092} C_VEL
LIN {X 0,Y 608.474,Z 82.812,A -85,B 0,C 180,E1 -488.587,E2 -488.587} C_VEL
LIN {X 0,Y 608.455,Z 82.814,A -85,B 0,C 180,E1 -491.341,E2 -491.341} C_VEL
LIN {X 0,Y 608.452,Z 82.816,A -85,B 0,C 180,E1 -494.263,E2 -494.263} C_VEL
LIN {X 0,Y 608.451,Z 82.814,A -85,B 0,C 180,E1 -497.04,E2 -497.04} C_VEL
LIN {X 0,Y 608.451,Z 82.822,A -85,B 0,C 180,E1 -499.697,E2 -499.697} C_VEL
LIN {X 0,Y 608.465,Z 82.812,A -85,B 0,C 180,E1 -502.253,E2 -502.253} C_VEL
LIN {X 0,Y 608.447,Z 82.818,A -85,B 0,C 180,E1 -505.094,E2 -505.094} C_VEL
LIN {X 0,Y 608.464,Z 82.814,A -85,B 0,C 180,E1 -507.905,E2 -507.905} C_VEL
LIN {X 0,Y 608.473,Z 82.81,A -85,B 0,C 180,E1 -510.221,E2 -510.221} C_VEL
LIN {X 0,Y 608.475,Z 82.814,A -85,B 0,C 180,E1 -512.793,E2 -512.793} C_VEL
LIN {X 0,Y 608.449,Z 82.818,A -85,B 0,C 180,E1 -515.429,E2 -515.429} C_VEL
LIN {X 0,Y 608.464,Z 82.812,A -85,B 0,C 180,E1 -518.308,E2 -518.308} C_VEL
LIN {X 0,Y 608.464,Z 82.816,A -85,B 0,C 180,E1 -521.285,E2 -521.285} C_VEL
LIN {X 0,Y 608.459,Z 82.812,A -85,B 0,C 180,E1 -523.906,E2 -523.906} C_VEL
LIN {X 0,Y 608.47,Z 82.819,A -85,B 0,C 180,E1 -526.644,E2 -526.644} C_VEL
LIN {X 0,Y 608.455,Z 82.813,A -85,B 0,C 180,E1 -529.35,E2 -529.35} C_VEL
LIN {X 0,Y 608.475,Z 82.812,A -85,B 0,C 180,E1 -532.033,E2 -532.033} C_VEL
LIN {X 0,Y 608.459,Z 82.819,A -85,B 0,C 180,E1 -534.698,E2 -534.698} C_VEL
LIN {X 0,Y 608.475,Z 82.81,A -85,B 0,C 180,E1 -537.352,E2 -537.352} C_VEL
LIN {X 0,Y 608.477,Z 82.815,A -85,B 0,C 180,E1 -540,E2 -540} C_VEL
LIN {X 0,Y 608.465,Z 82.815,A -85,B 0,C 180,E1 -542.648,E2 -542.648} C_VEL
LIN {X 0,Y 608.468,Z 82.811,A -85,B 0,C 180,E1 -545.302,E2 -545.302} C_VEL
LIN {X 0,Y 608.479,Z 82.819,A -85,B 0,C 180,E1 -547.967,E2 -547.967} C_VEL
LIN {X 0,Y 608.467,Z 82.813,A -85,B 0,C 180,E1 -549.445,E2 -549.445} C_VEL
LIN {X 0,Y 607.782,Z 82.907,A -85,B 0,C 180,E1 -549.998,E2 -549.998} C_VEL
LIN {X 0,Y 604.925,Z 83.264,A -85,B 0,C 180,E1 -550.895,E2 -550.895} C_VEL
LIN {X 0,Y 602.522,Z 83.561,A -85,B 0,C 180,E1 -551.616,E2 -551.616} C_VEL
LIN {X 0,Y 601.489,Z 83.686,A -85,B 0,C 180,E1 -552.173,E2 -552.173} C_VEL
LIN {X 0,Y 601.404,Z 83.694,A -85,B 0,C 180,E1 -552.361,E2 -552.361} C_VEL
LIN {X 0,Y 601.423,Z 83.688,A -85,B 0,C 180,E1 -554.897,E2 -554.897} C_VEL
LIN {X 0,Y 601.393,Z 83.702,A -85,B 0,C 180,E1 -557.689,E2 -557.689} C_VEL
LIN {X 0,Y 601.42,Z 83.689,A -85,B 0,C 180,E1 -560.522,E2 -560.522} C_VEL
LIN {X 0,Y 601.415,Z 83.698,A -85,B 0,C 180,E1 -563.411,E2 -563.411} C_VEL
LIN {X 0,Y 601.395,Z 83.692,A -85,B 0,C 180,E1 -566.364,E2 -566.364} C_VEL
LIN {X 0,Y 601.434,Z 83.689,A -85,B 0,C 180,E1 -568.789,E2 -568.789} C_VEL
LIN {X 0,Y 601.395,Z 83.695,A -85,B 0,C 180,E1 -571.728,E2 -571.728} C_VEL
LIN {X 0,Y 601.419,Z 83.689,A -85,B 0,C 180,E1 -574.119,E2 -574.119} C_VEL
LIN {X 0,Y 601.435,Z 83.692,A -85,B 0,C 180,E1 -577.382,E2 -577.382} C_VEL
LIN {X 0,Y 601.399,Z 83.691,A -85,B 0,C 180,E1 -579.996,E2 -579.996} C_VEL
LIN {X 0,Y 601.415,Z 83.696,A -85,B 0,C 180,E1 -582.67,E2 -582.67} C_VEL
LIN {X 0,Y 601.399,Z 83.692,A -85,B 0,C 180,E1 -585.48,E2 -585.48} C_VEL
LIN {X 0,Y 601.423,Z 83.694,A -85,B 0,C 180,E1 -588.407,E2 -588.407} C_VEL
LIN {X 0,Y 601.4,Z 83.697,A -85,B 0,C 180,E1 -590.873,E2 -590.873} C_VEL
LIN {X 0,Y 601.388,Z 83.693,A -85,B 0,C 180,E1 -593.416,E2 -593.416} C_VEL
LIN {X 0,Y 601.435,Z 83.691,A -85,B 0,C 180,E1 -596.065,E2 -596.065} C_VEL
LIN {X 0,Y 601.406,Z 83.691,A -85,B 0,C 180,E1 -599.057,E2 -599.057} C_VEL
LIN {X 0,Y 601.414,Z 83.69,A -85,B 0,C 180,E1 -601.372,E2 -601.372} C_VEL
LIN {X 0,Y 601.409,Z 83.697,A -85,B 0,C 180,E1 -604.382,E2 -604.382} C_VEL
LIN {X 0,Y 601.385,Z 83.696,A -85,B 0,C 180,E1 -606.588,E2 -606.588} C_VEL
LIN {X 0,Y 601.429,Z 83.69,A -85,B 0,C 180,E1 -609.478,E2 -609.478} C_VEL
LIN {X 0,Y 601.38,Z 83.698,A -85,B 0,C 180,E1 -612.311,E2 -612.311} C_VEL
LIN {X 0,Y 601.396,Z 83.707,A -85,B 0,C 180,E1 -614.886,E2 -614.886} C_VEL
LIN {X 0,Y 601.53,Z 92.41,A -85,B 0,C 180,E1 -616.166,E2 -616.166} C_VEL
LIN {X 0,Y 601.471,Z 108.833,A -85,B 0,C 180,E1 -618.543,E2 -618.543} C_VEL
LIN {X 0,Y 601.445,Z 119.534,A -85,B 0,C 180,E1 -620.075,E2 -620.075} C_VEL
LIN {X 0,Y 601.798,Z 121.426,A -85,B 0,C 180,E1 -620.124,E2 -620.124} C_VEL
LIN {X 0,Y 601.712,Z 256.464,A -85,B 0,C 180,E1 -621.774,E2 -621.774} C_VEL
LIN {X 0,Y 601.684,Z 270.88,A -85,B 0,C 180,E1 -622.09,E2 -622.09} C_VEL
LIN {X 0,Y 601.671,Z 284.672,A -85,B 0,C 180,E1 -622.533,E2 -622.533} C_VEL
LIN {X 0,Y 601.612,Z 297.188,A -85,B 0,C 180,E1 -623.064,E2 -623.064} C_VEL
LIN {X 0,Y 601.554,Z 310.165,A -85,B 0,C 180,E1 -623.763,E2 -623.763} C_VEL
LIN {X 0,Y 601.5,Z 321.99,A -85,B 0,C 180,E1 -624.553,E2 -624.553} C_VEL
LIN {X 0,Y 601.48,Z 333.344,A -85,B 0,C 180,E1 -625.476,E2 -625.476} C_VEL
LIN {X 0,Y 601.421,Z 343.554,A -85,B 0,C 180,E1 -626.483,E2 -626.483} C_VEL
LIN {X 0,Y 601.403,Z 352.009,A -85,B 0,C 180,E1 -627.488,E2 -627.488} C_VEL
LIN {X 0,Y 601.383,Z 360.124,A -85,B 0,C 180,E1 -628.661,E2 -628.661} C_VEL
LIN {X 0,Y 601.368,Z 365.836,A -85,B 0,C 180,E1 -629.665,E2 -629.665} C_VEL
LIN {X 0,Y 601.362,Z 370.523,A -85,B 0,C 180,E1 -630.67,E2 -630.67} C_VEL
LIN {X 0,Y 601.341,Z 375.396,A -85,B 0,C 180,E1 -632.009,E2 -632.009} C_VEL
LIN {X 0,Y 601.335,Z 378.799,A -85,B 0,C 180,E1 -633.35,E2 -633.35} C_VEL
LIN {X 0,Y 601.325,Z 380.816,A -85,B 0,C 180,E1 -634.693,E2 -634.693} C_VEL
LIN {X 0,Y 601.331,Z 381.5,A -85,B 0,C 180,E1 -636.038,E2 -636.038} C_VEL
LIN {X 0,Y 601.321,Z 380.828,A -85,B 0,C 180,E1 -637.387,E2 -637.387} C_VEL
LIN {X 0,Y 601.332,Z 378.8,A -85,B 0,C 180,E1 -638.739,E2 -638.739} C_VEL
LIN {X 0,Y 601.335,Z 375.345,A -85,B 0,C 180,E1 -640.097,E2 -640.097} C_VEL
LIN {X 0,Y 601.333,Z 370.355,A -85,B 0,C 180,E1 -641.46,E2 -641.46} C_VEL
LIN {X 0,Y 601.378,Z 365.506,A -85,B 0,C 180,E1 -642.486,E2 -642.486} C_VEL
LIN {X 0,Y 601.374,Z 359.584,A -85,B 0,C 180,E1 -643.517,E2 -643.517} C_VEL
LIN {X 0,Y 601.403,Z 352.387,A -85,B 0,C 180,E1 -644.552,E2 -644.552} C_VEL
LIN {X 0,Y 601.416,Z 343.7,A -85,B 0,C 180,E1 -645.591,E2 -645.591} C_VEL
LIN {X 0,Y 601.453,Z 333.173,A -85,B 0,C 180,E1 -646.629,E2 -646.629} C_VEL
LIN {X 0,Y 601.524,Z 322.37,A -85,B 0,C 180,E1 -647.509,E2 -647.509} C_VEL
LIN {X 0,Y 601.543,Z 310.611,A -85,B 0,C 180,E1 -648.3,E2 -648.3} C_VEL
LIN {X 0,Y 601.595,Z 298.041,A -85,B 0,C 180,E1 -648.984,E2 -648.984} C_VEL
LIN {X 0,Y 601.645,Z 285.258,A -85,B 0,C 180,E1 -649.535,E2 -649.535} C_VEL
LIN {X 0,Y 601.693,Z 271.652,A -85,B 0,C 180,E1 -649.978,E2 -649.978} C_VEL
LIN {X 0,Y 601.724,Z 257.916,A -85,B 0,C 180,E1 -650.288,E2 -650.288} C_VEL
LIN {X 0,Y 601.77,Z 228.424,A -85,B 0,C 180,E1 -650.67,E2 -650.67} C_VEL
LIN {X 0,Y 601.654,Z 120.82,A -85,B 0,C 180,E1 -651.978,E2 -651.978} C_VEL
LIN {X 0,Y 601.462,Z 119.62,A -85,B 0,C 180,E1 -652.002,E2 -652.002} C_VEL
LIN {X 0,Y 601.557,Z 100.766,A -85,B 0,C 180,E1 -654.709,E2 -654.709} C_VEL
LIN {X 0,Y 601.489,Z 84.329,A -85,B 0,C 180,E1 -657.109,E2 -657.109} C_VEL
LIN {X 0,Y 601.374,Z 83.698,A -85,B 0,C 180,E1 -657.242,E2 -657.242} C_VEL
LIN {X 0,Y 601.404,Z 83.701,A -85,B 0,C 180,E1 -660.165,E2 -660.165} C_VEL
LIN {X 0,Y 601.39,Z 83.694,A -85,B 0,C 180,E1 -662.71,E2 -662.71} C_VEL
LIN {X 0,Y 601.351,Z 83.698,A -85,B 0,C 180,E1 -665.105,E2 -665.105} C_VEL
LIN {X 0,Y 601.388,Z 83.696,A -85,B 0,C 180,E1 -667.422,E2 -667.422} C_VEL
LIN {X 0,Y 601.376,Z 83.701,A -85,B 0,C 180,E1 -669.998,E2 -669.998} C_VEL
LIN {X 0,Y 601.352,Z 83.698,A -85,B 0,C 180,E1 -672.584,E2 -672.584} C_VEL
LIN {X 0,Y 601.365,Z 83.696,A -85,B 0,C 180,E1 -674.529,E2 -674.529} C_VEL
LIN {X 0,Y 601.391,Z 83.701,A -85,B 0,C 180,E1 -677.412,E2 -677.412} C_VEL
LIN {X 0,Y 601.393,Z 83.693,A -85,B 0,C 180,E1 -680.003,E2 -680.003} C_VEL
LIN {X 0,Y 601.386,Z 83.694,A -85,B 0,C 180,E1 -682.624,E2 -682.624} C_VEL
LIN {X 0,Y 601.41,Z 83.697,A -85,B 0,C 180,E1 -685.067,E2 -685.067} C_VEL
LIN {X 0,Y 601.425,Z 83.693,A -85,B 0,C 180,E1 -687.484,E2 -687.484} C_VEL
LIN {X 0,Y 601.373,Z 83.695,A -85,B 0,C 180,E1 -689.861,E2 -689.861} C_VEL
LIN {X 0,Y 601.368,Z 83.696,A -85,B 0,C 180,E1 -692.13,E2 -692.13} C_VEL
LIN {X 0,Y 601.391,Z 83.695,A -85,B 0,C 180,E1 -694.38,E2 -694.38} C_VEL
LIN {X 0,Y 601.402,Z 83.693,A -85,B 0,C 180,E1 -697.316,E2 -697.316} C_VEL
LIN {X 0,Y 601.389,Z 83.696,A -85,B 0,C 180,E1 -700.19,E2 -700.19} C_VEL
LIN {X 0,Y 601.409,Z 83.694,A -85,B 0,C 180,E1 -703.013,E2 -703.013} C_VEL
LIN {X 0,Y 601.397,Z 83.693,A -85,B 0,C 180,E1 -705.794,E2 -705.794} C_VEL
LIN {X 0,Y 601.436,Z 83.694,A -85,B 0,C 180,E1 -708.542,E2 -708.542} C_VEL
LIN {X 0,Y 601.397,Z 83.691,A -85,B 0,C 180,E1 -711.262,E2 -711.262} C_VEL
LIN {X 0,Y 601.392,Z 83.693,A -85,B 0,C 180,E1 -713.378,E2 -713.378} C_VEL
LIN {X 0,Y 601.402,Z 83.699,A -85,B 0,C 180,E1 -715.979,E2 -715.979} C_VEL
LIN {X 0,Y 601.422,Z 83.69,A -85,B 0,C 180,E1 -718.661,E2 -718.661} C_VEL
LIN {X 0,Y 601.443,Z 83.686,A -85,B 0,C 180,E1 -720.669,E2 -720.669} C_VEL
LIN {X 0,Y 601.409,Z 83.693,A -85,B 0,C 180,E1 -723.35,E2 -723.35} C_VEL
LIN {X 0,Y 601.416,Z 83.694,A -85,B 0,C 180,E1 -726.037,E2 -726.037} C_VEL
LIN {X 0,Y 601.405,Z 83.691,A -85,B 0,C 180,E1 -728.738,E2 -728.738} C_VEL
LIN {X 0,Y 601.413,Z 83.699,A -85,B 0,C 180,E1 -731.458,E2 -731.458} C_VEL
LIN {X 0,Y 601.415,Z 83.69,A -85,B 0,C 180,E1 -734.205,E2 -734.205} C_VEL
LIN {X 0,Y 601.413,Z 83.694,A -85,B 0,C 180,E1 -736.986,E2 -736.986} C_VEL
LIN {X 0,Y 601.406,Z 83.692,A -85,B 0,C 180,E1 -739.809,E2 -739.809} C_VEL
LIN {X 0,Y 601.413,Z 83.693,A -85,B 0,C 180,E1 -742.683,E2 -742.683} C_VEL
LIN {X 0,Y 601.401,Z 83.699,A -85,B 0,C 180,E1 -744.879,E2 -744.879} C_VEL
LIN {X 0,Y 601.416,Z 83.693,A -85,B 0,C 180,E1 -747.363,E2 -747.363} C_VEL
LIN {X 0,Y 601.429,Z 83.689,A -85,B 0,C 180,E1 -750.164,E2 -750.164} C_VEL
LIN {X 0,Y 601.418,Z 83.699,A -85,B 0,C 180,E1 -752.715,E2 -752.715} C_VEL
LIN {X 0,Y 601.415,Z 83.692,A -85,B 0,C 180,E1 -755.115,E2 -755.115} C_VEL
LIN {X 0,Y 601.434,Z 83.687,A -85,B 0,C 180,E1 -757.419,E2 -757.419} C_VEL
LIN {X 0,Y 601.402,Z 83.693,A -85,B 0,C 180,E1 -759.996,E2 -759.996} C_VEL
LIN {X 0,Y 601.415,Z 83.695,A -85,B 0,C 180,E1 -762.67,E2 -762.67} C_VEL
LIN {X 0,Y 601.399,Z 83.692,A -85,B 0,C 180,E1 -765.479,E2 -765.479} C_VEL
LIN {X 0,Y 601.423,Z 83.695,A -85,B 0,C 180,E1 -768.407,E2 -768.407} C_VEL
LIN {X 0,Y 601.438,Z 83.687,A -85,B 0,C 180,E1 -770.875,E2 -770.875} C_VEL
LIN {X 0,Y 601.405,Z 83.693,A -85,B 0,C 180,E1 -773.417,E2 -773.417} C_VEL
LIN {X 0,Y 601.433,Z 83.694,A -85,B 0,C 180,E1 -776.064,E2 -776.064} C_VEL
LIN {X 0,Y 601.421,Z 83.689,A -85,B 0,C 180,E1 -778.545,E2 -778.545} C_VEL
LIN {X 0,Y 601.434,Z 83.692,A -85,B 0,C 180,E1 -781.373,E2 -781.373} C_VEL
LIN {X 0,Y 601.404,Z 83.701,A -85,B 0,C 180,E1 -783.636,E2 -783.636} C_VEL
LIN {X 0,Y 601.443,Z 83.734,A -85,B 0,C 180,E1 -786.385,E2 -786.385} C_VEL
LIN {X 0,Y 601.753,Z 86.699,A -85,B 0,C 180,E1 -786.786,E2 -786.786} C_VEL
LIN {X 0,Y 601.643,Z 109.027,A -85,B 0,C 180,E1 -789.664,E2 -789.664} C_VEL
LIN {X 0,Y 601.564,Z 131.355,A -85,B 0,C 180,E1 -792.492,E2 -792.492} C_VEL
LIN {X 0,Y 601.539,Z 143.697,A -85,B 0,C 180,E1 -794.037,E2 -794.037} C_VEL
LIN {X 0,Y 601.836,Z 147.608,A -85,B 0,C 180,E1 -794.094,E2 -794.094} C_VEL
LIN {X 0,Y 601.716,Z 281.977,A -85,B 0,C 180,E1 -795.739,E2 -795.739} C_VEL
LIN {X 0,Y 601.716,Z 296.11,A -85,B 0,C 180,E1 -796.053,E2 -796.053} C_VEL
LIN {X 0,Y 601.636,Z 309.711,A -85,B 0,C 180,E1 -796.489,E2 -796.489} C_VEL
LIN {X 0,Y 601.6,Z 323.633,A -85,B 0,C 180,E1 -797.09,E2 -797.09} C_VEL
LIN {X 0,Y 601.543,Z 336.093,A -85,B 0,C 180,E1 -797.774,E2 -797.774} C_VEL
LIN {X 0,Y 601.504,Z 347.472,A -85,B 0,C 180,E1 -798.543,E2 -798.543} C_VEL
LIN {X 0,Y 601.482,Z 357.931,A -85,B 0,C 180,E1 -799.395,E2 -799.395} C_VEL
LIN {X 0,Y 601.43,Z 368.333,A -85,B 0,C 180,E1 -800.414,E2 -800.414} C_VEL
LIN {X 0,Y 601.407,Z 376.913,A -85,B 0,C 180,E1 -801.431,E2 -801.431} C_VEL
LIN {X 0,Y 601.392,Z 385.113,A -85,B 0,C 180,E1 -802.614,E2 -802.614} C_VEL
LIN {X 0,Y 601.361,Z 390.751,A -85,B 0,C 180,E1 -803.604,E2 -803.604} C_VEL
LIN {X 0,Y 601.354,Z 395.567,A -85,B 0,C 180,E1 -804.635,E2 -804.635} C_VEL
LIN {X 0,Y 601.345,Z 400.441,A -85,B 0,C 180,E1 -805.979,E2 -805.979} C_VEL
LIN {X 0,Y 601.322,Z 403.831,A -85,B 0,C 180,E1 -807.32,E2 -807.32} C_VEL
LIN {X 0,Y 601.342,Z 405.831,A -85,B 0,C 180,E1 -808.661,E2 -808.661} C_VEL
LIN {X 0,Y 601.333,Z 406.5,A -85,B 0,C 180,E1 -810,E2 -810} C_VEL
LIN {X 0,Y 601.342,Z 405.831,A -85,B 0,C 180,E1 -811.339,E2 -811.339} C_VEL
LIN {X 0,Y 601.322,Z 403.832,A -85,B 0,C 180,E1 -812.679,E2 -812.679} C_VEL
LIN {X 0,Y 601.345,Z 400.443,A -85,B 0,C 180,E1 -814.021,E2 -814.021} C_VEL
LIN {X 0,Y 601.354,Z 395.568,A -85,B 0,C 180,E1 -815.365,E2 -815.365} C_VEL
LIN {X 0,Y 601.372,Z 389.623,A -85,B 0,C 180,E1 -816.605,E2 -816.605} C_VEL
LIN {X 0,Y 601.386,Z 382.92,A -85,B 0,C 180,E1 -817.723,E2 -817.723} C_VEL
LIN {X 0,Y 601.411,Z 374.199,A -85,B 0,C 180,E1 -818.907,E2 -818.907} C_VEL
LIN {X 0,Y 601.433,Z 365.083,A -85,B 0,C 180,E1 -819.925,E2 -819.925} C_VEL
LIN {X 0,Y 601.497,Z 354.829,A -85,B 0,C 180,E1 -820.876,E2 -820.876} C_VEL
LIN {X 0,Y 601.533,Z 343.972,A -85,B 0,C 180,E1 -821.712,E2 -821.712} C_VEL
LIN {X 0,Y 601.575,Z 331.78,A -85,B 0,C 180,E1 -822.482,E2 -822.482} C_VEL
LIN {X 0,Y 601.619,Z 320.096,A -85,B 0,C 180,E1 -823.081,E2 -823.081} C_VEL
LIN {X 0,Y 601.657,Z 307.94,A -85,B 0,C 180,E1 -823.578,E2 -823.578} C_VEL
LIN {X 0,Y 601.709,Z 294.033,A -85,B 0,C 180,E1 -824.004,E2 -824.004} C_VEL
LIN {X 0,Y 601.736,Z 279.906,A -85,B 0,C 180,E1 -824.295,E2 -824.295} C_VEL
LIN {X 0,Y 601.739,Z 144.946,A -85,B 0,C 180,E1 -825.941,E2 -825.941} C_VEL
LIN {X 0,Y 601.539,Z 143.568,A -85,B 0,C 180,E1 -825.979,E2 -825.979} C_VEL
LIN {X 0,Y 601.598,Z 122.495,A -85,B 0,C 180,E1 -828.624,E2 -828.624} C_VEL
LIN {X 0,Y 601.695,Z 99.261,A -85,B 0,C 180,E1 -831.588,E2 -831.588} C_VEL
LIN {X 0,Y 601.746,Z 85.306,A -85,B 0,C 180,E1 -833.397,E2 -833.397} C_VEL
LIN {X 0,Y 601.426,Z 83.693,A -85,B 0,C 180,E1 -833.638,E2 -833.638} C_VEL
LIN {X 0,Y 601.403,Z 83.701,A -85,B 0,C 180,E1 -836.364,E2 -836.364} C_VEL
LIN {X 0,Y 601.439,Z 83.69,A -85,B 0,C 180,E1 -838.789,E2 -838.789} C_VEL
LIN {X 0,Y 601.42,Z 83.69,A -85,B 0,C 180,E1 -841.454,E2 -841.454} C_VEL
LIN {X 0,Y 601.429,Z 83.697,A -85,B 0,C 180,E1 -844.118,E2 -844.118} C_VEL
LIN {X 0,Y 601.436,Z 83.688,A -85,B 0,C 180,E1 -847.382,E2 -847.382} C_VEL
LIN {X 0,Y 601.41,Z 83.7,A -85,B 0,C 180,E1 -849.995,E2 -849.995} C_VEL
LIN {X 0,Y 601.409,Z 83.691,A -85,B 0,C 180,E1 -852.67,E2 -852.67} C_VEL
LIN {X 0,Y 601.426,Z 83.693,A -85,B 0,C 180,E1 -855.482,E2 -855.482} C_VEL
LIN {X 0,Y 601.424,Z 83.689,A -85,B 0,C 180,E1 -858.407,E2 -858.407} C_VEL
LIN {X 0,Y 601.429,Z 83.697,A -85,B 0,C 180,E1 -861.529,E2 -861.529} C_VEL
LIN {X 0,Y 601.388,Z 83.693,A -85,B 0,C 180,E1 -864.245,E2 -864.245} C_VEL
LIN {X 0,Y 601.427,Z 83.689,A -85,B 0,C 180,E1 -866.686,E2 -866.686} C_VEL
LIN {X 0,Y 601.419,Z 83.694,A -85,B 0,C 180,E1 -869.058,E2 -869.058} C_VEL
LIN {X 0,Y 601.43,Z 83.696,A -85,B 0,C 180,E1 -871.373,E2 -871.373} C_VEL
LIN {X 0,Y 601.415,Z 83.689,A -85,B 0,C 180,E1 -874.132,E2 -874.132} C_VEL
LIN {X 0,Y 601.418,Z 83.692,A -85,B 0,C 180,E1 -876.59,E2 -876.59} C_VEL
LIN {X 0,Y 601.425,Z 83.691,A -85,B 0,C 180,E1 -879.478,E2 -879.478} C_VEL
LIN {X 0,Y 601.399,Z 83.693,A -85,B 0,C 180,E1 -882.312,E2 -882.312} C_VEL
LIN {X 0,Y 601.417,Z 83.693,A -85,B 0,C 180,E1 -884.409,E2 -884.409} C_VEL
LIN {X 0,Y 601.418,Z 83.692,A -85,B 0,C 180,E1 -887.172,E2 -887.172} C_VEL
LIN {X 0,Y 601.43,Z 83.688,A -85,B 0,C 180,E1 -889.905,E2 -889.905} C_VEL
LIN {X 0,Y 601.438,Z 83.696,A -85,B 0,C 180,E1 -892.615,E2 -892.615} C_VEL
LIN {X 0,Y 601.419,Z 83.689,A -85,B 0,C 180,E1 -895.308,E2 -895.308} C_VEL
LIN {X 0,Y 601.426,Z 83.692,A -85,B 0,C 180,E1 -897.991,E2 -897.991} C_VEL
LIN {X 0,Y 601.441,Z 83.69,A -85,B 0,C 180,E1 -900.67,E2 -900.67} C_VEL
LIN {X 0,Y 601.429,Z 83.688,A -85,B 0,C 180,E1 -903.35,E2 -903.35} C_VEL
LIN {X 0,Y 601.41,Z 83.699,A -85,B 0,C 180,E1 -906.037,E2 -906.037} C_VEL
LIN {X 0,Y 601.439,Z 83.697,A -85,B 0,C 180,E1 -908.061,E2 -908.061} C_VEL
LIN {X 0,Y 601.418,Z 83.689,A -85,B 0,C 180,E1 -911.01,E2 -911.01} C_VEL
LIN {X 0,Y 601.404,Z 83.694,A -85,B 0,C 180,E1 -912.361,E2 -912.361} C_VEL
LIN {X 0,Y 600.736,Z 83.777,A -85,B 0,C 180,E1 -912.921,E2 -912.921} C_VEL
LIN {X 0,Y 597.887,Z 84.139,A -85,B 0,C 180,E1 -913.829,E2 -913.829} C_VEL
LIN {X 0,Y 595.479,Z 84.433,A -85,B 0,C 180,E1 -914.559,E2 -914.559} C_VEL
LIN {X 0,Y 594.444,Z 84.559,A -85,B 0,C 180,E1 -915.122,E2 -915.122} C_VEL
LIN {X 0,Y 594.358,Z 84.571,A -85,B 0,C 180,E1 -915.313,E2 -915.313} C_VEL
LIN {X 0,Y 594.344,Z 84.577,A -85,B 0,C 180,E1 -917.905,E2 -917.905} C_VEL
LIN {X 0,Y 594.397,Z 84.564,A -85,B 0,C 180,E1 -920.776,E2 -920.776} C_VEL
LIN {X 0,Y 594.381,Z 84.573,A -85,B 0,C 180,E1 -923.705,E2 -923.705} C_VEL
LIN {X 0,Y 594.382,Z 84.566,A -85,B 0,C 180,E1 -926.7,E2 -926.7} C_VEL
LIN {X 0,Y 594.379,Z 84.57,A -85,B 0,C 180,E1 -928.999,E2 -928.999} C_VEL
LIN {X 0,Y 594.374,Z 84.571,A -85,B 0,C 180,E1 -931.642,E2 -931.642} C_VEL
LIN {X 0,Y 594.378,Z 84.568,A -85,B 0,C 180,E1 -934.58,E2 -934.58} C_VEL
LIN {X 0,Y 594.387,Z 84.567,A -85,B 0,C 180,E1 -937.608,E2 -937.608} C_VEL
LIN {X 0,Y 594.366,Z 84.571,A -85,B 0,C 180,E1 -940.568,E2 -940.568} C_VEL
LIN {X 0,Y 594.353,Z 84.573,A -85,B 0,C 180,E1 -943.301,E2 -943.301} C_VEL
LIN {X 0,Y 594.362,Z 84.57,A -85,B 0,C 180,E1 -946.162,E2 -946.162} C_VEL
LIN {X 0,Y 594.37,Z 84.57,A -85,B 0,C 180,E1 -949.179,E2 -949.179} C_VEL
LIN {X 0,Y 594.379,Z 84.568,A -85,B 0,C 180,E1 -952.059,E2 -952.059} C_VEL
LIN {X 0,Y 594.348,Z 84.577,A -85,B 0,C 180,E1 -954.678,E2 -954.678} C_VEL
LIN {X 0,Y 594.376,Z 84.567,A -85,B 0,C 180,E1 -957.089,E2 -957.089} C_VEL
LIN {X 0,Y 594.387,Z 84.566,A -85,B 0,C 180,E1 -959.672,E2 -959.672} C_VEL
LIN {X 0,Y 594.341,Z 84.576,A -85,B 0,C 180,E1 -962.538,E2 -962.538} C_VEL
LIN {X 0,Y 594.359,Z 84.57,A -85,B 0,C 180,E1 -964.806,E2 -964.806} C_VEL
LIN {X 0,Y 594.362,Z 84.568,A -85,B 0,C 180,E1 -967.266,E2 -967.266} C_VEL
LIN {X 0,Y 594.368,Z 84.577,A -85,B 0,C 180,E1 -969.946,E2 -969.946} C_VEL
LIN {X 0,Y 594.372,Z 84.568,A -85,B 0,C 180,E1 -972.806,E2 -972.806} C_VEL
LIN {X 0,Y 594.39,Z 84.679,A -85,B 0,C 180,E1 -974.769,E2 -974.769} C_VEL
LIN {X 0,Y 594.644,Z 90.408,A -85,B 0,C 180,E1 -975.629,E2 -975.629} C_VEL
LIN {X 0,Y 594.489,Z 109.354,A -85,B 0,C 180,E1 -978.406,E2 -978.406} C_VEL
LIN {X 0,Y 594.454,Z 119.606,A -85,B 0,C 180,E1 -979.893,E2 -979.893} C_VEL
LIN {X 0,Y 594.985,Z 123.868,A -85,B 0,C 180,E1 -979.966,E2 -979.966} C_VEL
LIN {X 0,Y 594.839,Z 256.916,A -85,B 0,C 180,E1 -981.614,E2 -981.614} C_VEL
LIN {X 0,Y 594.799,Z 271.178,A -85,B 0,C 180,E1 -981.934,E2 -981.934} C_VEL
LIN {X 0,Y 594.759,Z 285.449,A -85,B 0,C 180,E1 -982.404,E2 -982.404} C_VEL
LIN {X 0,Y 594.663,Z 299.007,A -85,B 0,C 180,E1 -983,E2 -983} C_VEL
LIN {X 0,Y 594.585,Z 311.23,A -85,B 0,C 180,E1 -983.682,E2 -983.682} C_VEL
LIN {X 0,Y 594.504,Z 322.971,A -85,B 0,C 180,E1 -984.488,E2 -984.488} C_VEL
LIN {X 0,Y 594.467,Z 334.161,A -85,B 0,C 180,E1 -985.423,E2 -985.423} C_VEL
LIN {X 0,Y 594.374,Z 344.197,A -85,B 0,C 180,E1 -986.441,E2 -986.441} C_VEL
LIN {X 0,Y 594.343,Z 352.547,A -85,B 0,C 180,E1 -987.459,E2 -987.459} C_VEL
LIN {X 0,Y 594.299,Z 360.554,A -85,B 0,C 180,E1 -988.645,E2 -988.645} C_VEL
LIN {X 0,Y 594.299,Z 366.216,A -85,B 0,C 180,E1 -989.661,E2 -989.661} C_VEL
LIN {X 0,Y 594.267,Z 370.825,A -85,B 0,C 180,E1 -990.678,E2 -990.678} C_VEL
LIN {X 0,Y 594.241,Z 375.622,A -85,B 0,C 180,E1 -992.033,E2 -992.033} C_VEL
LIN {X 0,Y 594.255,Z 378.952,A -85,B 0,C 180,E1 -993.39,E2 -993.39} C_VEL
LIN {X 0,Y 594.224,Z 380.896,A -85,B 0,C 180,E1 -994.749,E2 -994.749} C_VEL
LIN {X 0,Y 594.236,Z 381.491,A -85,B 0,C 180,E1 -996.11,E2 -996.11} C_VEL
LIN {X 0,Y 594.246,Z 380.746,A -85,B 0,C 180,E1 -997.475,E2 -997.475} C_VEL
LIN {X 0,Y 594.229,Z 378.646,A -85,B 0,C 180,E1 -998.845,E2 -998.845} C_VEL
LIN {X 0,Y 594.247,Z 375.117,A -85,B 0,C 180,E1 -1000.219,E2 -1000.219} C_VEL
LIN {X 0,Y 594.27,Z 370.049,A -85,B 0,C 180,E1 -1001.598,E2 -1001.598} C_VEL
LIN {X 0,Y 594.288,Z 365.112,A -85,B 0,C 180,E1 -1002.637,E2 -1002.637} C_VEL
LIN {X 0,Y 594.325,Z 357.562,A -85,B 0,C 180,E1 -1003.915,E2 -1003.915} C_VEL
LIN {X 0,Y 594.337,Z 349.043,A -85,B 0,C 180,E1 -1005.079,E2 -1005.079} C_VEL
LIN {X 0,Y 594.425,Z 339.67,A -85,B 0,C 180,E1 -1006.132,E2 -1006.132} C_VEL
LIN {X 0,Y 594.46,Z 330.021,A -85,B 0,C 180,E1 -1007.035,E2 -1007.035} C_VEL
LIN {X 0,Y 594.543,Z 318.94,A -85,B 0,C 180,E1 -1007.899,E2 -1007.899} C_VEL
LIN {X 0,Y 594.62,Z 306.286,A -85,B 0,C 180,E1 -1008.703,E2 -1008.703} C_VEL
LIN {X 0,Y 594.682,Z 293.133,A -85,B 0,C 180,E1 -1009.369,E2 -1009.369} C_VEL
LIN {X 0,Y 594.779,Z 279.387,A -85,B 0,C 180,E1 -1009.905,E2 -1009.905} C_VEL
LIN {X 0,Y 594.796,Z 265.096,A -85,B 0,C 180,E1 -1010.309,E2 -1010.309} C_VEL
LIN {X 0,Y 594.851,Z 251.654,A -85,B 0,C 180,E1 -1010.556,E2 -1010.556} C_VEL
LIN {X 0,Y 594.956,Z 122.277,A -85,B 0,C 180,E1 -1012.144,E2 -1012.144} C_VEL
LIN {X 0,Y 594.467,Z 119.539,A -85,B 0,C 180,E1 -1012.207,E2 -1012.207} C_VEL
LIN {X 0,Y 594.578,Z 100.479,A -85,B 0,C 180,E1 -1014.978,E2 -1014.978} C_VEL
LIN {X 0,Y 594.569,Z 86.318,A -85,B 0,C 180,E1 -1017.07,E2 -1017.07} C_VEL
LIN {X 0,Y 594.325,Z 84.578,A -85,B 0,C 180,E1 -1017.368,E2 -1017.368} C_VEL
LIN {X 0,Y 594.365,Z 84.576,A -85,B 0,C 180,E1 -1020.324,E2 -1020.324} C_VEL
LIN {X 0,Y 594.337,Z 84.572,A -85,B 0,C 180,E1 -1022.953,E2 -1022.953} C_VEL
LIN {X 0,Y 594.307,Z 84.577,A -85,B 0,C 180,E1 -1025.412,E2 -1025.412} C_VEL
LIN {X 0,Y 594.347,Z 84.579,A -85,B 0,C 180,E1 -1027.944,E2 -1027.944} C_VEL
LIN {X 0,Y 594.331,Z 84.572,A -85,B 0,C 180,E1 -1030.816,E2 -1030.816} C_VEL
LIN {X 0,Y 594.336,Z 84.576,A -85,B 0,C 180,E1 -1033.302,E2 -1033.302} C_VEL
LIN {X 0,Y 594.341,Z 84.572,A -85,B 0,C 180,E1 -1036.163,E2 -1036.163} C_VEL
LIN {X 0,Y 594.354,Z 84.569,A -85,B 0,C 180,E1 -1038.534,E2 -1038.534} C_VEL
LIN {X 0,Y 594.362,Z 84.576,A -85,B 0,C 180,E1 -1041.298,E2 -1041.298} C_VEL
LIN {X 0,Y 594.342,Z 84.573,A -85,B 0,C 180,E1 -1043.755,E2 -1043.755} C_VEL
LIN {X 0,Y 594.349,Z 84.57,A -85,B 0,C 180,E1 -1046.237,E2 -1046.237} C_VEL
LIN {X 0,Y 594.359,Z 84.572,A -85,B 0,C 180,E1 -1048.649,E2 -1048.649} C_VEL
LIN {X 0,Y 594.38,Z 84.576,A -85,B 0,C 180,E1 -1051.043,E2 -1051.043} C_VEL
LIN {X 0,Y 594.35,Z 84.569,A -85,B 0,C 180,E1 -1053.985,E2 -1053.985} C_VEL
LIN {X 0,Y 594.346,Z 84.573,A -85,B 0,C 180,E1 -1056.294,E2 -1056.294} C_VEL
LIN {X 0,Y 594.392,Z 84.567,A -85,B 0,C 180,E1 -1059.224,E2 -1059.224} C_VEL
LIN {X 0,Y 594.335,Z 84.574,A -85,B 0,C 180,E1 -1062.094,E2 -1062.094} C_VEL
LIN {X 0,Y 594.354,Z 84.574,A -85,B 0,C 180,E1 -1064.219,E2 -1064.219} C_VEL
LIN {X 0,Y 594.351,Z 84.571,A -85,B 0,C 180,E1 -1067.016,E2 -1067.016} C_VEL
LIN {X 0,Y 594.359,Z 84.569,A -85,B 0,C 180,E1 -1069.094,E2 -1069.094} C_VEL
LIN {X 0,Y 594.377,Z 84.569,A -85,B 0,C 180,E1 -1071.843,E2 -1071.843} C_VEL
LIN {X 0,Y 594.394,Z 84.567,A -85,B 0,C 180,E1 -1074.572,E2 -1074.572} C_VEL
LIN {X 0,Y 594.385,Z 84.566,A -85,B 0,C 180,E1 -1077.289,E2 -1077.289} C_VEL
LIN {X 0,Y 594.416,Z 84.57,A -85,B 0,C 180,E1 -1080,E2 -1080} C_VEL
LIN {X 0,Y 594.402,Z 84.563,A -85,B 0,C 180,E1 -1082.711,E2 -1082.711} C_VEL
LIN {X 0,Y 594.378,Z 84.571,A -85,B 0,C 180,E1 -1085.428,E2 -1085.428} C_VEL
LIN {X 0,Y 594.413,Z 84.564,A -85,B 0,C 180,E1 -1088.157,E2 -1088.157} C_VEL
LIN {X 0,Y 594.381,Z 84.568,A -85,B 0,C 180,E1 -1091.069,E2 -1091.069} C_VEL
LIN {X 0,Y 594.38,Z 84.572,A -85,B 0,C 180,E1 -1093.679,E2 -1093.679} C_VEL
LIN {X 0,Y 594.368,Z 84.568,A -85,B 0,C 180,E1 -1096.711,E2 -1096.711} C_VEL
LIN {X 0,Y 594.368,Z 84.575,A -85,B 0,C 180,E1 -1099.334,E2 -1099.334} C_VEL
LIN {X 0,Y 594.359,Z 84.573,A -85,B 0,C 180,E1 -1101.504,E2 -1101.504} C_VEL
LIN {X 0,Y 594.389,Z 84.566,A -85,B 0,C 180,E1 -1104.446,E2 -1104.446} C_VEL
LIN {X 0,Y 594.383,Z 84.571,A -85,B 0,C 180,E1 -1106.7,E2 -1106.7} C_VEL
LIN {X 0,Y 594.381,Z 84.574,A -85,B 0,C 180,E1 -1108.998,E2 -1108.998} C_VEL
LIN {X 0,Y 594.391,Z 84.565,A -85,B 0,C 180,E1 -1111.645,E2 -1111.645} C_VEL
LIN {X 0,Y 594.396,Z 84.573,A -85,B 0,C 180,E1 -1114.579,E2 -1114.579} C_VEL
LIN {X 0,Y 594.388,Z 84.565,A -85,B 0,C 180,E1 -1117.608,E2 -1117.608} C_VEL
LIN {X 0,Y 594.369,Z 84.575,A -85,B 0,C 180,E1 -1120.567,E2 -1120.567} C_VEL
LIN {X 0,Y 594.369,Z 84.567,A -85,B 0,C 180,E1 -1123.299,E2 -1123.299} C_VEL
LIN {X 0,Y 594.361,Z 84.577,A -85,B 0,C 180,E1 -1126.161,E2 -1126.161} C_VEL
LIN {X 0,Y 594.38,Z 84.57,A -85,B 0,C 180,E1 -1128.536,E2 -1128.536} C_VEL
LIN {X 0,Y 594.39,Z 84.565,A -85,B 0,C 180,E1 -1131.295,E2 -1131.295} C_VEL
LIN {X 0,Y 594.354,Z 84.576,A -85,B 0,C 180,E1 -1133.756,E2 -1133.756} C_VEL
LIN {X 0,Y 594.377,Z 84.57,A -85,B 0,C 180,E1 -1136.239,E2 -1136.239} C_VEL
LIN {X 0,Y 594.371,Z 84.567,A -85,B 0,C 180,E1 -1138.65,E2 -1138.65} C_VEL
LIN {X 0,Y 594.385,Z 84.567,A -85,B 0,C 180,E1 -1141.042,E2 -1141.042} C_VEL
LIN {X 0,Y 594.383,Z 84.571,A -85,B 0,C 180,E1 -1143.978,E2 -1143.978} C_VEL
LIN {X 0,Y 594.397,Z 84.606,A -85,B 0,C 180,E1 -1146.204,E2 -1146.204} C_VEL
LIN {X 0,Y 594.892,Z 88.095,A -85,B 0,C 180,E1 -1146.686,E2 -1146.686} C_VEL
LIN {X 0,Y 594.729,Z 110.423,A -85,B 0,C 180,E1 -1149.598,E2 -1149.598} C_VEL
LIN {X 0,Y 594.6,Z 132.751,A -85,B 0,C 180,E1 -1152.458,E2 -1152.458} C_VEL
LIN {X 0,Y 594.522,Z 143.566,A -85,B 0,C 180,E1 -1153.827,E2 -1153.827} C_VEL
LIN {X 0,Y 595.022,Z 147.608,A -85,B 0,C 180,E1 -1153.907,E2 -1153.907} C_VEL
LIN {X 0,Y 594.856,Z 281.88,A -85,B 0,C 180,E1 -1155.569,E2 -1155.569} C_VEL
LIN {X 0,Y 594.809,Z 296.176,A -85,B 0,C 180,E1 -1155.889,E2 -1155.889} C_VEL
LIN {X 0,Y 594.716,Z 309.711,A -85,B 0,C 180,E1 -1156.329,E2 -1156.329} C_VEL
LIN {X 0,Y 594.647,Z 323.636,A -85,B 0,C 180,E1 -1156.936,E2 -1156.936} C_VEL
LIN {X 0,Y 594.58,Z 336.095,A -85,B 0,C 180,E1 -1157.629,E2 -1157.629} C_VEL
LIN {X 0,Y 594.524,Z 348.559,A -85,B 0,C 180,E1 -1158.488,E2 -1158.488} C_VEL
LIN {X 0,Y 594.449,Z 359.835,A -85,B 0,C 180,E1 -1159.441,E2 -1159.441} C_VEL
LIN {X 0,Y 594.368,Z 369.85,A -85,B 0,C 180,E1 -1160.471,E2 -1160.471} C_VEL
LIN {X 0,Y 594.324,Z 378.17,A -85,B 0,C 180,E1 -1161.5,E2 -1161.5} C_VEL
LIN {X 0,Y 594.303,Z 386.125,A -85,B 0,C 180,E1 -1162.696,E2 -1162.696} C_VEL
LIN {X 0,Y 594.281,Z 392.527,A -85,B 0,C 180,E1 -1163.89,E2 -1163.89} C_VEL
LIN {X 0,Y 594.236,Z 398.199,A -85,B 0,C 180,E1 -1165.251,E2 -1165.251} C_VEL
LIN {X 0,Y 594.258,Z 402.315,A -85,B 0,C 180,E1 -1166.61,E2 -1166.61} C_VEL
LIN {X 0,Y 594.242,Z 405,A -85,B 0,C 180,E1 -1167.967,E2 -1167.967} C_VEL
LIN {X 0,Y 594.234,Z 406.332,A -85,B 0,C 180,E1 -1169.322,E2 -1169.322} C_VEL
LIN {X 0,Y 594.234,Z 406.332,A -85,B 0,C 180,E1 -1170.678,E2 -1170.678} C_VEL
LIN {X 0,Y 594.242,Z 405.001,A -85,B 0,C 180,E1 -1172.033,E2 -1172.033} C_VEL
LIN {X 0,Y 594.258,Z 402.317,A -85,B 0,C 180,E1 -1173.39,E2 -1173.39} C_VEL
LIN {X 0,Y 594.236,Z 398.2,A -85,B 0,C 180,E1 -1174.749,E2 -1174.749} C_VEL
LIN {X 0,Y 594.281,Z 392.527,A -85,B 0,C 180,E1 -1176.11,E2 -1176.11} C_VEL
LIN {X 0,Y 594.303,Z 386.127,A -85,B 0,C 180,E1 -1177.303,E2 -1177.303} C_VEL
LIN {X 0,Y 594.323,Z 378.171,A -85,B 0,C 180,E1 -1178.5,E2 -1178.5} C_VEL
LIN {X 0,Y 594.367,Z 369.852,A -85,B 0,C 180,E1 -1179.529,E2 -1179.529} C_VEL
LIN {X 0,Y 594.449,Z 359.837,A -85,B 0,C 180,E1 -1180.559,E2 -1180.559} C_VEL
LIN {X 0,Y 594.524,Z 348.565,A -85,B 0,C 180,E1 -1181.512,E2 -1181.512} C_VEL
LIN {X 0,Y 594.58,Z 336.1,A -85,B 0,C 180,E1 -1182.371,E2 -1182.371} C_VEL
LIN {X 0,Y 594.645,Z 323.642,A -85,B 0,C 180,E1 -1183.064,E2 -1183.064} C_VEL
LIN {X 0,Y 594.713,Z 309.713,A -85,B 0,C 180,E1 -1183.671,E2 -1183.671} C_VEL
LIN {X 0,Y 594.814,Z 295.623,A -85,B 0,C 180,E1 -1184.126,E2 -1184.126} C_VEL
LIN {X 0,Y 594.858,Z 281.891,A -85,B 0,C 180,E1 -1184.431,E2 -1184.431} C_VEL
LIN {X 0,Y 594.922,Z 145.838,A -85,B 0,C 180,E1 -1186.118,E2 -1186.118} C_VEL
LIN {X 0,Y 594.522,Z 143.568,A -85,B 0,C 180,E1 -1186.173,E2 -1186.173} C_VEL
LIN {X 0,Y 594.648,Z 123.32,A -85,B 0,C 180,E1 -1188.744,E2 -1188.744} C_VEL
LIN {X 0,Y 594.746,Z 102.052,A -85,B 0,C 180,E1 -1191.489,E2 -1191.489} C_VEL
LIN {X 0,Y 594.822,Z 86.701,A -85,B 0,C 180,E1 -1193.501,E2 -1193.501} C_VEL
LIN {X 0,Y 594.389,Z 84.57,A -85,B 0,C 180,E1 -1193.82,E2 -1193.82} C_VEL
LIN {X 0,Y 594.386,Z 84.571,A -85,B 0,C 180,E1 -1196.699,E2 -1196.699} C_VEL
LIN {X 0,Y 594.382,Z 84.567,A -85,B 0,C 180,E1 -1198.998,E2 -1198.998} C_VEL
LIN {X 0,Y 594.378,Z 84.568,A -85,B 0,C 180,E1 -1201.642,E2 -1201.642} C_VEL
LIN {X 0,Y 594.381,Z 84.569,A -85,B 0,C 180,E1 -1204.58,E2 -1204.58} C_VEL
LIN {X 0,Y 594.39,Z 84.568,A -85,B 0,C 180,E1 -1207.608,E2 -1207.608} C_VEL
LIN {X 0,Y 594.37,Z 84.569,A -85,B 0,C 180,E1 -1210.567,E2 -1210.567} C_VEL
LIN {X 0,Y 594.365,Z 84.57,A -85,B 0,C 180,E1 -1213.299,E2 -1213.299} C_VEL
LIN {X 0,Y 594.383,Z 84.569,A -85,B 0,C 180,E1 -1216.159,E2 -1216.159} C_VEL
LIN {X 0,Y 594.377,Z 84.569,A -85,B 0,C 180,E1 -1219.178,E2 -1219.178} C_VEL
LIN {X 0,Y 594.383,Z 84.568,A -85,B 0,C 180,E1 -1222.059,E2 -1222.059} C_VEL
LIN {X 0,Y 594.353,Z 84.569,A -85,B 0,C 180,E1 -1224.676,E2 -1224.676} C_VEL
LIN {X 0,Y 594.378,Z 84.571,A -85,B 0,C 180,E1 -1227.088,E2 -1227.088} C_VEL
LIN {X 0,Y 594.385,Z 84.569,A -85,B 0,C 180,E1 -1229.672,E2 -1229.672} C_VEL
LIN {X 0,Y 594.374,Z 84.568,A -85,B 0,C 180,E1 -1232.539,E2 -1232.539} C_VEL
LIN {X 0,Y 594.376,Z 84.571,A -85,B 0,C 180,E1 -1234.807,E2 -1234.807} C_VEL
LIN {X 0,Y 594.364,Z 84.574,A -85,B 0,C 180,E1 -1237.265,E2 -1237.265} C_VEL
LIN {X 0,Y 594.372,Z 84.567,A -85,B 0,C 180,E1 -1239.946,E2 -1239.946} C_VEL
LIN {X 0,Y 594.38,Z 84.575,A -85,B 0,C 180,E1 -1242.806,E2 -1242.806} C_VEL
LIN {X 0,Y 594.388,Z 84.565,A -85,B 0,C 180,E1 -1245.826,E2 -1245.826} C_VEL
LIN {X 0,Y 594.393,Z 84.569,A -85,B 0,C 180,E1 -1248.404,E2 -1248.404} C_VEL
LIN {X 0,Y 594.379,Z 84.568,A -85,B 0,C 180,E1 -1251.158,E2 -1251.158} C_VEL
LIN {X 0,Y 594.364,Z 84.569,A -85,B 0,C 180,E1 -1253.891,E2 -1253.891} C_VEL
LIN {X 0,Y 594.375,Z 84.573,A -85,B 0,C 180,E1 -1256.611,E2 -1256.611} C_VEL
LIN {X 0,Y 594.418,Z 84.561,A -85,B 0,C 180,E1 -1259.323,E2 -1259.323} C_VEL
LIN {X 0,Y 594.394,Z 84.571,A -85,B 0,C 180,E1 -1262.033,E2 -1262.033} C_VEL
LIN {X 0,Y 594.383,Z 84.567,A -85,B 0,C 180,E1 -1264.748,E2 -1264.748} C_VEL
LIN {X 0,Y 594.394,Z 84.566,A -85,B 0,C 180,E1 -1267.473,E2 -1267.473} C_VEL
LIN {X 0,Y 594.389,Z 84.571,A -85,B 0,C 180,E1 -1270.216,E2 -1270.216} C_VEL
LIN {X 0,Y 594.362,Z 84.568,A -85,B 0,C 180,E1 -1272.983,E2 -1272.983} C_VEL
LIN {X 0,Y 594.358,Z 84.571,A -85,B 0,C 180,E1 -1275.313,E2 -1275.313} C_VEL
LIN {X 0,Y 593.684,Z 84.661,A -85,B 0,C 180,E1 -1275.879,E2 -1275.879} C_VEL
LIN {X 0,Y 590.814,Z 85.021,A -85,B 0,C 180,E1 -1276.797,E2 -1276.797} C_VEL
LIN {X 0,Y 588.4,Z 85.318,A -85,B 0,C 180,E1 -1277.535,E2 -1277.535} C_VEL
LIN {X 0,Y 587.377,Z 85.442,A -85,B 0,C 180,E1 -1278.105,E2 -1278.105} C_VEL
LIN {X 0,Y 587.3,Z 85.449,A -85,B 0,C 180,E1 -1278.298,E2 -1278.298} C_VEL
LIN {X 0,Y 587.33,Z 85.446,A -85,B 0,C 180,E1 -1281.038,E2 -1281.038} C_VEL
LIN {X 0,Y 587.319,Z 85.451,A -85,B 0,C 180,E1 -1283.259,E2 -1283.259} C_VEL
LIN {X 0,Y 587.331,Z 85.453,A -85,B 0,C 180,E1 -1285.517,E2 -1285.517} C_VEL
LIN {X 0,Y 587.345,Z 85.445,A -85,B 0,C 180,E1 -1287.818,E2 -1287.818} C_VEL
LIN {X 0,Y 587.322,Z 85.445,A -85,B 0,C 180,E1 -1290.508,E2 -1290.508} C_VEL
LIN {X 0,Y 587.336,Z 85.452,A -85,B 0,C 180,E1 -1293.112,E2 -1293.112} C_VEL
LIN {X 0,Y 587.289,Z 85.45,A -85,B 0,C 180,E1 -1295.9,E2 -1295.9} C_VEL
LIN {X 0,Y 587.322,Z 85.447,A -85,B 0,C 180,E1 -1298.48,E2 -1298.48} C_VEL
LIN {X 0,Y 587.333,Z 85.45,A -85,B 0,C 180,E1 -1301.158,E2 -1301.158} C_VEL
LIN {X 0,Y 587.318,Z 85.446,A -85,B 0,C 180,E1 -1304.113,E2 -1304.113} C_VEL
LIN {X 0,Y 587.299,Z 85.454,A -85,B 0,C 180,E1 -1306.992,E2 -1306.992} C_VEL
LIN {X 0,Y 587.308,Z 85.447,A -85,B 0,C 180,E1 -1309.745,E2 -1309.745} C_VEL
LIN {X 0,Y 587.342,Z 85.449,A -85,B 0,C 180,E1 -1312.392,E2 -1312.392} C_VEL
LIN {X 0,Y 587.356,Z 85.442,A -85,B 0,C 180,E1 -1315.78,E2 -1315.78} C_VEL
LIN {X 0,Y 587.337,Z 85.451,A -85,B 0,C 180,E1 -1318.231,E2 -1318.231} C_VEL
LIN {X 0,Y 587.346,Z 85.444,A -85,B 0,C 180,E1 -1320.868,E2 -1320.868} C_VEL
LIN {X 0,Y 587.31,Z 85.451,A -85,B 0,C 180,E1 -1323.83,E2 -1323.83} C_VEL
LIN {X 0,Y 587.329,Z 85.452,A -85,B 0,C 180,E1 -1325.993,E2 -1325.993} C_VEL
LIN {X 0,Y 587.317,Z 85.453,A -85,B 0,C 180,E1 -1328.226,E2 -1328.226} C_VEL
LIN {X 0,Y 587.346,Z 85.443,A -85,B 0,C 180,E1 -1331.151,E2 -1331.151} C_VEL
LIN {X 0,Y 587.311,Z 85.456,A -85,B 0,C 180,E1 -1334.025,E2 -1334.025} C_VEL
LIN {X 0,Y 587.36,Z 85.654,A -85,B 0,C 180,E1 -1334.649,E2 -1334.649} C_VEL
LIN {X 0,Y 587.702,Z 89.753,A -85,B 0,C 180,E1 -1335.279,E2 -1335.279} C_VEL
LIN {X 0,Y 587.526,Z 108.688,A -85,B 0,C 180,E1 -1338.092,E2 -1338.092} C_VEL
LIN {X 0,Y 587.433,Z 119.533,A -85,B 0,C 180,E1 -1339.684,E2 -1339.684} C_VEL
LIN {X 0,Y 588.164,Z 124.575,A -85,B 0,C 180,E1 -1339.784,E2 -1339.784} C_VEL
LIN {X 0,Y 587.983,Z 256.222,A -85,B 0,C 180,E1 -1341.429,E2 -1341.429} C_VEL
LIN {X 0,Y 587.914,Z 269.986,A -85,B 0,C 180,E1 -1341.731,E2 -1341.731} C_VEL
LIN {X 0,Y 587.862,Z 284.01,A -85,B 0,C 180,E1 -1342.184,E2 -1342.184} C_VEL
LIN {X 0,Y 587.779,Z 296.152,A -85,B 0,C 180,E1 -1342.702,E2 -1342.702} C_VEL
LIN {X 0,Y 587.658,Z 308.684,A -85,B 0,C 180,E1 -1343.377,E2 -1343.377} C_VEL
LIN {X 0,Y 587.558,Z 320.508,A -85,B 0,C 180,E1 -1344.165,E2 -1344.165} C_VEL
LIN {X 0,Y 587.451,Z 331.156,A -85,B 0,C 180,E1 -1345.024,E2 -1345.024} C_VEL
LIN {X 0,Y 587.361,Z 341.719,A -85,B 0,C 180,E1 -1346.055,E2 -1346.055} C_VEL
LIN {X 0,Y 587.308,Z 350.477,A -85,B 0,C 180,E1 -1347.085,E2 -1347.085} C_VEL
LIN {X 0,Y 587.285,Z 358.895,A -85,B 0,C 180,E1 -1348.286,E2 -1348.286} C_VEL
LIN {X 0,Y 587.201,Z 364.806,A -85,B 0,C 180,E1 -1349.314,E2 -1349.314} C_VEL
LIN {X 0,Y 587.172,Z 371.128,A -85,B 0,C 180,E1 -1350.686,E2 -1350.686} C_VEL
LIN {X 0,Y 587.141,Z 375.849,A -85,B 0,C 180,E1 -1352.058,E2 -1352.058} C_VEL
LIN {X 0,Y 587.178,Z 379.097,A -85,B 0,C 180,E1 -1353.431,E2 -1353.431} C_VEL
LIN {X 0,Y 587.123,Z 380.955,A -85,B 0,C 180,E1 -1354.807,E2 -1354.807} C_VEL
LIN {X 0,Y 587.147,Z 381.475,A -85,B 0,C 180,E1 -1356.184,E2 -1356.184} C_VEL
LIN {X 0,Y 587.145,Z 380.662,A -85,B 0,C 180,E1 -1357.566,E2 -1357.566} C_VEL
LIN {X 0,Y 587.129,Z 378.492,A -85,B 0,C 180,E1 -1358.952,E2 -1358.952} C_VEL
LIN {X 0,Y 587.169,Z 374.889,A -85,B 0,C 180,E1 -1360.343,E2 -1360.343} C_VEL
LIN {X 0,Y 587.187,Z 369.74,A -85,B 0,C 180,E1 -1361.74,E2 -1361.74} C_VEL
LIN {X 0,Y 587.2,Z 364.717,A -85,B 0,C 180,E1 -1362.793,E2 -1362.793} C_VEL
LIN {X 0,Y 587.243,Z 358.612,A -85,B 0,C 180,E1 -1363.849,E2 -1363.849} C_VEL
LIN {X 0,Y 587.282,Z 349.839,A -85,B 0,C 180,E1 -1365.087,E2 -1365.087} C_VEL
LIN {X 0,Y 587.381,Z 340.622,A -85,B 0,C 180,E1 -1366.152,E2 -1366.152} C_VEL
LIN {X 0,Y 587.463,Z 329.456,A -85,B 0,C 180,E1 -1367.217,E2 -1367.217} C_VEL
LIN {X 0,Y 587.59,Z 317.838,A -85,B 0,C 180,E1 -1368.118,E2 -1368.118} C_VEL
LIN {X 0,Y 587.653,Z 306.581,A -85,B 0,C 180,E1 -1368.839,E2 -1368.839} C_VEL
LIN {X 0,Y 587.752,Z 293.929,A -85,B 0,C 180,E1 -1369.493,E2 -1369.493} C_VEL
LIN {X 0,Y 587.899,Z 281.128,A -85,B 0,C 180,E1 -1370.011,E2 -1370.011} C_VEL
LIN {X 0,Y 587.907,Z 267.543,A -85,B 0,C 180,E1 -1370.421,E2 -1370.421} C_VEL
LIN {X 0,Y 587.985,Z 252.585,A -85,B 0,C 180,E1 -1370.715,E2 -1370.715} C_VEL
LIN {X 0,Y 588.15,Z 123.164,A -85,B 0,C 180,E1 -1372.324,E2 -1372.324} C_VEL
LIN {X 0,Y 587.513,Z 119.622,A -85,B 0,C 180,E1 -1372.391,E2 -1372.391} C_VEL
LIN {X 0,Y 587.612,Z 99.789,A -85,B 0,C 180,E1 -1375.314,E2 -1375.314} C_VEL
LIN {X 0,Y 587.557,Z 87.052,A -85,B 0,C 180,E1 -1377.223,E2 -1377.223} C_VEL
LIN {X 0,Y 587.284,Z 85.456,A -85,B 0,C 180,E1 -1377.493,E2 -1377.493} C_VEL
LIN {X 0,Y 587.31,Z 85.457,A -85,B 0,C 180,E1 -1380.172,E2 -1380.172} C_VEL
LIN {X 0,Y 587.285,Z 85.45,A -85,B 0,C 180,E1 -1383.103,E2 -1383.103} C_VEL
LIN {X 0,Y 587.26,Z 85.457,A -85,B 0,C 180,E1 -1385.532,E2 -1385.532} C_VEL
LIN {X 0,Y 587.304,Z 85.457,A -85,B 0,C 180,E1 -1387.833,E2 -1387.833} C_VEL
LIN {X 0,Y 587.286,Z 85.453,A -85,B 0,C 180,E1 -1390.257,E2 -1390.257} C_VEL
LIN {X 0,Y 587.277,Z 85.453,A -85,B 0,C 180,E1 -1393.114,E2 -1393.114} C_VEL
LIN {X 0,Y 587.298,Z 85.451,A -85,B 0,C 180,E1 -1396.047,E2 -1396.047} C_VEL
LIN {X 0,Y 587.3,Z 85.45,A -85,B 0,C 180,E1 -1398.929,E2 -1398.929} C_VEL
LIN {X 0,Y 587.308,Z 85.454,A -85,B 0,C 180,E1 -1401.519,E2 -1401.519} C_VEL
LIN {X 0,Y 587.279,Z 85.451,A -85,B 0,C 180,E1 -1404.099,E2 -1404.099} C_VEL
LIN {X 0,Y 587.319,Z 85.447,A -85,B 0,C 180,E1 -1406.602,E2 -1406.602} C_VEL
LIN {X 0,Y 587.313,Z 85.456,A -85,B 0,C 180,E1 -1409.032,E2 -1409.032} C_VEL
LIN {X 0,Y 587.302,Z 85.451,A -85,B 0,C 180,E1 -1411.402,E2 -1411.402} C_VEL
LIN {X 0,Y 587.305,Z 85.447,A -85,B 0,C 180,E1 -1413.83,E2 -1413.83} C_VEL
LIN {X 0,Y 587.3,Z 85.457,A -85,B 0,C 180,E1 -1416.74,E2 -1416.74} C_VEL
LIN {X 0,Y 587.315,Z 85.446,A -85,B 0,C 180,E1 -1419.694,E2 -1419.694} C_VEL
LIN {X 0,Y 587.289,Z 85.449,A -85,B 0,C 180,E1 -1421.872,E2 -1421.872} C_VEL
LIN {X 0,Y 587.307,Z 85.45,A -85,B 0,C 180,E1 -1424.024,E2 -1424.024} C_VEL
LIN {X 0,Y 587.302,Z 85.451,A -85,B 0,C 180,E1 -1426.858,E2 -1426.858} C_VEL
LIN {X 0,Y 587.329,Z 85.446,A -85,B 0,C 180,E1 -1429.66,E2 -1429.66} C_VEL
LIN {X 0,Y 587.362,Z 85.447,A -85,B 0,C 180,E1 -1432.437,E2 -1432.437} C_VEL
LIN {X 0,Y 587.344,Z 85.442,A -85,B 0,C 180,E1 -1435.195,E2 -1435.195} C_VEL
LIN {X 0,Y 587.371,Z 85.447,A -85,B 0,C 180,E1 -1437.943,E2 -1437.943} C_VEL
LIN {X 0,Y 587.386,Z 85.437,A -85,B 0,C 180,E1 -1440.685,E2 -1440.685} C_VEL
LIN {X 0,Y 587.315,Z 85.45,A -85,B 0,C 180,E1 -1443.43,E2 -1443.43} C_VEL
LIN {X 0,Y 587.345,Z 85.448,A -85,B 0,C 180,E1 -1445.493,E2 -1445.493} C_VEL
LIN {X 0,Y 587.364,Z 85.442,A -85,B 0,C 180,E1 -1448.255,E2 -1448.255} C_VEL
LIN {X 0,Y 587.35,Z 85.445,A -85,B 0,C 180,E1 -1451.134,E2 -1451.134} C_VEL
LIN {X 0,Y 587.341,Z 85.443,A -85,B 0,C 180,E1 -1454.251,E2 -1454.251} C_VEL
LIN {X 0,Y 587.346,Z 85.45,A -85,B 0,C 180,E1 -1457.406,E2 -1457.406} C_VEL
LIN {X 0,Y 587.324,Z 85.444,A -85,B 0,C 180,E1 -1460.305,E2 -1460.305} C_VEL
LIN {X 0,Y 587.315,Z 85.453,A -85,B 0,C 180,E1 -1463.259,E2 -1463.259} C_VEL
LIN {X 0,Y 587.336,Z 85.446,A -85,B 0,C 180,E1 -1465.517,E2 -1465.517} C_VEL
LIN {X 0,Y 587.347,Z 85.442,A -85,B 0,C 180,E1 -1467.818,E2 -1467.818} C_VEL
LIN {X 0,Y 587.342,Z 85.447,A -85,B 0,C 180,E1 -1470.511,E2 -1470.511} C_VEL
LIN {X 0,Y 587.336,Z 85.445,A -85,B 0,C 180,E1 -1473.397,E2 -1473.397} C_VEL
LIN {X 0,Y 587.294,Z 85.449,A -85,B 0,C 180,E1 -1475.9,E2 -1475.9} C_VEL
LIN {X 0,Y 587.326,Z 85.454,A -85,B 0,C 180,E1 -1478.48,E2 -1478.48} C_VEL
LIN {X 0,Y 587.337,Z 85.444,A -85,B 0,C 180,E1 -1481.157,E2 -1481.157} C_VEL
LIN {X 0,Y 587.328,Z 85.451,A -85,B 0,C 180,E1 -1484.113,E2 -1484.113} C_VEL
LIN {X 0,Y 587.314,Z 85.447,A -85,B 0,C 180,E1 -1486.993,E2 -1486.993} C_VEL
LIN {X 0,Y 587.318,Z 85.45,A -85,B 0,C 180,E1 -1489.746,E2 -1489.746} C_VEL
LIN {X 0,Y 587.346,Z 85.446,A -85,B 0,C 180,E1 -1492.392,E2 -1492.392} C_VEL
LIN {X 0,Y 587.363,Z 85.448,A -85,B 0,C 180,E1 -1495.78,E2 -1495.78} C_VEL
LIN {X 0,Y 587.342,Z 85.446,A -85,B 0,C 180,E1 -1498.231,E2 -1498.231} C_VEL
LIN {X 0,Y 587.351,Z 85.443,A -85,B 0,C 180,E1 -1500.867,E2 -1500.867} C_VEL
LIN {X 0,Y 587.359,Z 85.448,A -85,B 0,C 180,E1 -1503.819,E2 -1503.819} C_VEL
LIN {X 0,Y 587.369,Z 85.518,A -85,B 0,C 180,E1 -1506.042,E2 -1506.042} C_VEL
LIN {X 0,Y 588,Z 89.411,A -85,B 0,C 180,E1 -1506.583,E2 -1506.583} C_VEL
LIN {X 0,Y 587.795,Z 111.818,A -85,B 0,C 180,E1 -1509.529,E2 -1509.529} C_VEL
LIN {X 0,Y 587.631,Z 134.146,A -85,B 0,C 180,E1 -1512.423,E2 -1512.423} C_VEL
LIN {X 0,Y 587.578,Z 143.809,A -85,B 0,C 180,E1 -1513.65,E2 -1513.65} C_VEL
LIN {X 0,Y 588.208,Z 147.608,A -85,B 0,C 180,E1 -1513.715,E2 -1513.715} C_VEL
LIN {X 0,Y 587.992,Z 281.88,A -85,B 0,C 180,E1 -1515.397,E2 -1515.397} C_VEL
LIN {X 0,Y 587.926,Z 296.29,A -85,B 0,C 180,E1 -1515.724,E2 -1515.724} C_VEL
LIN {X 0,Y 587.802,Z 310.837,A -85,B 0,C 180,E1 -1516.209,E2 -1516.209} C_VEL
LIN {X 0,Y 587.725,Z 323.639,A -85,B 0,C 180,E1 -1516.78,E2 -1516.78} C_VEL
LIN {X 0,Y 587.604,Z 336.098,A -85,B 0,C 180,E1 -1517.48,E2 -1517.48} C_VEL
LIN {X 0,Y 587.513,Z 347.477,A -85,B 0,C 180,E1 -1518.266,E2 -1518.266} C_VEL
LIN {X 0,Y 587.465,Z 357.934,A -85,B 0,C 180,E1 -1519.139,E2 -1519.139} C_VEL
LIN {X 0,Y 587.353,Z 368.333,A -85,B 0,C 180,E1 -1520.182,E2 -1520.182} C_VEL
LIN {X 0,Y 587.311,Z 376.912,A -85,B 0,C 180,E1 -1521.224,E2 -1521.224} C_VEL
LIN {X 0,Y 587.249,Z 385.115,A -85,B 0,C 180,E1 -1522.435,E2 -1522.435} C_VEL
LIN {X 0,Y 587.18,Z 391.68,A -85,B 0,C 180,E1 -1523.635,E2 -1523.635} C_VEL
LIN {X 0,Y 587.158,Z 396.961,A -85,B 0,C 180,E1 -1524.849,E2 -1524.849} C_VEL
LIN {X 0,Y 587.181,Z 400.442,A -85,B 0,C 180,E1 -1525.882,E2 -1525.882} C_VEL
LIN {X 0,Y 587.129,Z 403.831,A -85,B 0,C 180,E1 -1527.255,E2 -1527.255} C_VEL
LIN {X 0,Y 587.142,Z 405.832,A -85,B 0,C 180,E1 -1528.628,E2 -1528.628} C_VEL
LIN {X 0,Y 587.135,Z 406.5,A -85,B 0,C 180,E1 -1530,E2 -1530} C_VEL
LIN {X 0,Y 587.142,Z 405.833,A -85,B 0,C 180,E1 -1531.372,E2 -1531.372} C_VEL
LIN {X 0,Y 587.129,Z 403.833,A -85,B 0,C 180,E1 -1532.744,E2 -1532.744} C_VEL
LIN {X 0,Y 587.181,Z 400.444,A -85,B 0,C 180,E1 -1534.118,E2 -1534.118} C_VEL
LIN {X 0,Y 587.199,Z 395.568,A -85,B 0,C 180,E1 -1535.494,E2 -1535.494} C_VEL
LIN {X 0,Y 587.209,Z 389.053,A -85,B 0,C 180,E1 -1536.874,E2 -1536.874} C_VEL
LIN {X 0,Y 587.268,Z 381.801,A -85,B 0,C 180,E1 -1538.083,E2 -1538.083} C_VEL
LIN {X 0,Y 587.321,Z 372.824,A -85,B 0,C 180,E1 -1539.296,E2 -1539.296} C_VEL
LIN {X 0,Y 587.372,Z 363.393,A -85,B 0,C 180,E1 -1540.339,E2 -1540.339} C_VEL
LIN {X 0,Y 587.475,Z 353.03,A -85,B 0,C 180,E1 -1541.29,E2 -1541.29} C_VEL
LIN {X 0,Y 587.577,Z 341.434,A -85,B 0,C 180,E1 -1542.17,E2 -1542.17} C_VEL
LIN {X 0,Y 587.664,Z 328.648,A -85,B 0,C 180,E1 -1542.958,E2 -1542.958} C_VEL
LIN {X 0,Y 587.773,Z 316.159,A -85,B 0,C 180,E1 -1543.571,E2 -1543.571} C_VEL
LIN {X 0,Y 587.902,Z 302.729,A -85,B 0,C 180,E1 -1544.081,E2 -1544.081} C_VEL
LIN {X 0,Y 587.962,Z 288.306,A -85,B 0,C 180,E1 -1544.477,E2 -1544.477} C_VEL
LIN {X 0,Y 588.01,Z 274.612,A -85,B 0,C 180,E1 -1544.713,E2 -1544.713} C_VEL
LIN {X 0,Y 588.13,Z 146.733,A -85,B 0,C 180,E1 -1546.298,E2 -1546.298} C_VEL
LIN {X 0,Y 587.565,Z 143.568,A -85,B 0,C 180,E1 -1546.37,E2 -1546.37} C_VEL
LIN {X 0,Y 587.691,Z 124.38,A -85,B 0,C 180,E1 -1548.837,E2 -1548.837} C_VEL
LIN {X 0,Y 587.834,Z 104.764,A -85,B 0,C 180,E1 -1551.396,E2 -1551.396} C_VEL
LIN {X 0,Y 587.999,Z 89.414,A -85,B 0,C 180,E1 -1553.417,E2 -1553.417} C_VEL
LIN {X 0,Y 587.364,Z 85.446,A -85,B 0,C 180,E1 -1553.982,E2 -1553.982} C_VEL
LIN {X 0,Y 587.331,Z 85.446,A -85,B 0,C 180,E1 -1557.046,E2 -1557.046} C_VEL
LIN {X 0,Y 587.346,Z 85.443,A -85,B 0,C 180,E1 -1559.379,E2 -1559.379} C_VEL
LIN {X 0,Y 587.345,Z 85.447,A -85,B 0,C 180,E1 -1561.835,E2 -1561.835} C_VEL
LIN {X 0,Y 587.349,Z 85.448,A -85,B 0,C 180,E1 -1564.348,E2 -1564.348} C_VEL
LIN {X 0,Y 587.346,Z 85.445,A -85,B 0,C 180,E1 -1567.607,E2 -1567.607} C_VEL
LIN {X 0,Y 587.318,Z 85.451,A -85,B 0,C 180,E1 -1570.254,E2 -1570.254} C_VEL
LIN {X 0,Y 587.314,Z 85.447,A -85,B 0,C 180,E1 -1573.118,E2 -1573.118} C_VEL
LIN {X 0,Y 587.335,Z 85.449,A -85,B 0,C 180,E1 -1576.051,E2 -1576.051} C_VEL
LIN {X 0,Y 587.336,Z 85.444,A -85,B 0,C 180,E1 -1578.925,E2 -1578.925} C_VEL
LIN {X 0,Y 587.327,Z 85.454,A -85,B 0,C 180,E1 -1581.52,E2 -1581.52} C_VEL
LIN {X 0,Y 587.291,Z 85.45,A -85,B 0,C 180,E1 -1584.1,E2 -1584.1} C_VEL
LIN {X 0,Y 587.335,Z 85.444,A -85,B 0,C 180,E1 -1586.603,E2 -1586.603} C_VEL
LIN {X 0,Y 587.337,Z 85.45,A -85,B 0,C 180,E1 -1589.49,E2 -1589.49} C_VEL
LIN {X 0,Y 587.35,Z 85.442,A -85,B 0,C 180,E1 -1592.307,E2 -1592.307} C_VEL
LIN {X 0,Y 587.336,Z 85.444,A -85,B 0,C 180,E1 -1594.483,E2 -1594.483} C_VEL
LIN {X 0,Y 587.338,Z 85.446,A -85,B 0,C 180,E1 -1597.486,E2 -1597.486} C_VEL
LIN {X 0,Y 587.313,Z 85.448,A -85,B 0,C 180,E1 -1600.424,E2 -1600.424} C_VEL
LIN {X 0,Y 587.327,Z 85.448,A -85,B 0,C 180,E1 -1603.311,E2 -1603.311} C_VEL
LIN {X 0,Y 587.361,Z 85.442,A -85,B 0,C 180,E1 -1606.154,E2 -1606.154} C_VEL
LIN {X 0,Y 587.336,Z 85.448,A -85,B 0,C 180,E1 -1608.962,E2 -1608.962} C_VEL
LIN {X 0,Y 587.364,Z 85.44,A -85,B 0,C 180,E1 -1611.745,E2 -1611.745} C_VEL
LIN {X 0,Y 587.353,Z 85.451,A -85,B 0,C 180,E1 -1614.507,E2 -1614.507} C_VEL
LIN {X 0,Y 587.372,Z 85.439,A -85,B 0,C 180,E1 -1617.257,E2 -1617.257} C_VEL
LIN {X 0,Y 587.383,Z 85.442,A -85,B 0,C 180,E1 -1620,E2 -1620} C_VEL
LIN {X 0,Y 587.366,Z 85.442,A -85,B 0,C 180,E1 -1622.743,E2 -1622.743} C_VEL
LIN {X 0,Y 587.359,Z 85.442,A -85,B 0,C 180,E1 -1625.493,E2 -1625.493} C_VEL
LIN {X 0,Y 587.363,Z 85.446,A -85,B 0,C 180,E1 -1628.255,E2 -1628.255} C_VEL
LIN {X 0,Y 587.348,Z 85.442,A -85,B 0,C 180,E1 -1631.134,E2 -1631.134} C_VEL
LIN {X 0,Y 587.365,Z 85.443,A -85,B 0,C 180,E1 -1634.261,E2 -1634.261} C_VEL
LIN {X 0,Y 587.34,Z 85.447,A -85,B 0,C 180,E1 -1637.406,E2 -1637.406} C_VEL
LIN {X 0,Y 587.3,Z 85.449,A -85,B 0,C 180,E1 -1638.298,E2 -1638.298} C_VEL
LIN {X 0,Y 586.66,Z 85.528,A -85,B 0,C 180,E1 -1638.87,E2 -1638.87} C_VEL
LIN {X 0,Y 583.841,Z 85.886,A -85,B 0,C 180,E1 -1639.799,E2 -1639.799} C_VEL
LIN {X 0,Y 581.433,Z 86.188,A -85,B 0,C 180,E1 -1640.546,E2 -1640.546} C_VEL
LIN {X 0,Y 580.378,Z 86.317,A -85,B 0,C 180,E1 -1641.123,E2 -1641.123} C_VEL
LIN {X 0,Y 580.282,Z 86.327,A -85,B 0,C 180,E1 -1641.318,E2 -1641.318} C_VEL
LIN {X 0,Y 580.272,Z 86.333,A -85,B 0,C 180,E1 -1643.558,E2 -1643.558} C_VEL
LIN {X 0,Y 580.28,Z 86.326,A -85,B 0,C 180,E1 -1645.85,E2 -1645.85} C_VEL
LIN {X 0,Y 580.297,Z 86.321,A -85,B 0,C 180,E1 -1648.186,E2 -1648.186} C_VEL
LIN {X 0,Y 580.273,Z 86.325,A -85,B 0,C 180,E1 -1650.693,E2 -1650.693} C_VEL
LIN {X 0,Y 580.283,Z 86.33,A -85,B 0,C 180,E1 -1653.314,E2 -1653.314} C_VEL
LIN {X 0,Y 580.244,Z 86.328,A -85,B 0,C 180,E1 -1655.756,E2 -1655.756} C_VEL
LIN {X 0,Y 580.285,Z 86.322,A -85,B 0,C 180,E1 -1658.147,E2 -1658.147} C_VEL
LIN {X 0,Y 580.296,Z 86.328,A -85,B 0,C 180,E1 -1660.844,E2 -1660.844} C_VEL
LIN {X 0,Y 580.27,Z 86.324,A -85,B 0,C 180,E1 -1663.659,E2 -1663.659} C_VEL
LIN {X 0,Y 580.268,Z 86.331,A -85,B 0,C 180,E1 -1666.611,E2 -1666.611} C_VEL
LIN {X 0,Y 580.296,Z 86.323,A -85,B 0,C 180,E1 -1669.157,E2 -1669.157} C_VEL
LIN {X 0,Y 580.287,Z 86.323,A -85,B 0,C 180,E1 -1671.928,E2 -1671.928} C_VEL
LIN {X 0,Y 580.25,Z 86.335,A -85,B 0,C 180,E1 -1674.453,E2 -1674.453} C_VEL
LIN {X 0,Y 580.29,Z 86.323,A -85,B 0,C 180,E1 -1676.975,E2 -1676.975} C_VEL
LIN {X 0,Y 580.295,Z 86.32,A -85,B 0,C 180,E1 -1679.425,E2 -1679.425} C_VEL
LIN {X 0,Y 580.257,Z 86.333,A -85,B 0,C 180,E1 -1682.15,E2 -1682.15} C_VEL
LIN {X 0,Y 580.322,Z 86.317,A -85,B 0,C 180,E1 -1685.271,E2 -1685.271} C_VEL
LIN {X 0,Y 580.269,Z 86.332,A -85,B 0,C 180,E1 -1687.947,E2 -1687.947} C_VEL
LIN {X 0,Y 580.296,Z 86.322,A -85,B 0,C 180,E1 -1690.913,E2 -1690.913} C_VEL
LIN {X 0,Y 580.265,Z 86.335,A -85,B 0,C 180,E1 -1693.825,E2 -1693.825} C_VEL
LIN {X 0,Y 580.299,Z 86.432,A -85,B 0,C 180,E1 -1694.48,E2 -1694.48} C_VEL
LIN {X 0,Y 580.776,Z 90.329,A -85,B 0,C 180,E1 -1695.099,E2 -1695.099} C_VEL
LIN {X 0,Y 580.539,Z 109.21,A -85,B 0,C 180,E1 -1697.946,E2 -1697.946} C_VEL
LIN {X 0,Y 580.503,Z 119.915,A -85,B 0,C 180,E1 -1699.504,E2 -1699.504} C_VEL
LIN {X 0,Y 581.357,Z 125.276,A -85,B 0,C 180,E1 -1699.597,E2 -1699.597} C_VEL
LIN {X 0,Y 581.128,Z 256.685,A -85,B 0,C 180,E1 -1701.262,E2 -1701.262} C_VEL
LIN {X 0,Y 581.031,Z 271.032,A -85,B 0,C 180,E1 -1701.589,E2 -1701.589} C_VEL
LIN {X 0,Y 580.95,Z 284.79,A -85,B 0,C 180,E1 -1702.047,E2 -1702.047} C_VEL
LIN {X 0,Y 580.832,Z 297.633,A -85,B 0,C 180,E1 -1702.614,E2 -1702.614} C_VEL
LIN {X 0,Y 580.69,Z 309.615,A -85,B 0,C 180,E1 -1703.28,E2 -1703.28} C_VEL
LIN {X 0,Y 580.575,Z 321.493,A -85,B 0,C 180,E1 -1704.094,E2 -1704.094} C_VEL
LIN {X 0,Y 580.421,Z 331.98,A -85,B 0,C 180,E1 -1704.964,E2 -1704.964} C_VEL
LIN {X 0,Y 580.32,Z 342.407,A -85,B 0,C 180,E1 -1706.007,E2 -1706.007} C_VEL
LIN {X 0,Y 580.244,Z 351.05,A -85,B 0,C 180,E1 -1707.049,E2 -1707.049} C_VEL
LIN {X 0,Y 580.226,Z 359.366,A -85,B 0,C 180,E1 -1708.265,E2 -1708.265} C_VEL
LIN {X 0,Y 580.113,Z 365.19,A -85,B 0,C 180,E1 -1709.306,E2 -1709.306} C_VEL
LIN {X 0,Y 580.077,Z 371.43,A -85,B 0,C 180,E1 -1710.694,E2 -1710.694} C_VEL
LIN {X 0,Y 580.041,Z 376.065,A -85,B 0,C 180,E1 -1712.083,E2 -1712.083} C_VEL
LIN {X 0,Y 580.104,Z 379.22,A -85,B 0,C 180,E1 -1713.473,E2 -1713.473} C_VEL
LIN {X 0,Y 580.026,Z 381.005,A -85,B 0,C 180,E1 -1714.866,E2 -1714.866} C_VEL
LIN {X 0,Y 580.065,Z 381.458,A -85,B 0,C 180,E1 -1716.26,E2 -1716.26} C_VEL
LIN {X 0,Y 580.065,Z 380.58,A -85,B 0,C 180,E1 -1717.659,E2 -1717.659} C_VEL
LIN {X 0,Y 580.029,Z 378.337,A -85,B 0,C 180,E1 -1719.063,E2 -1719.063} C_VEL
LIN {X 0,Y 580.092,Z 374.66,A -85,B 0,C 180,E1 -1720.471,E2 -1720.471} C_VEL
LIN {X 0,Y 580.115,Z 369.432,A -85,B 0,C 180,E1 -1721.885,E2 -1721.885} C_VEL
LIN {X 0,Y 580.147,Z 364.324,A -85,B 0,C 180,E1 -1722.951,E2 -1722.951} C_VEL
LIN {X 0,Y 580.19,Z 358.125,A -85,B 0,C 180,E1 -1724.02,E2 -1724.02} C_VEL
LIN {X 0,Y 580.247,Z 349.246,A -85,B 0,C 180,E1 -1725.274,E2 -1725.274} C_VEL
LIN {X 0,Y 580.38,Z 339.911,A -85,B 0,C 180,E1 -1726.352,E2 -1726.352} C_VEL
LIN {X 0,Y 580.467,Z 329.54,A -85,B 0,C 180,E1 -1727.346,E2 -1727.346} C_VEL
LIN {X 0,Y 580.621,Z 318.031,A -85,B 0,C 180,E1 -1728.252,E2 -1728.252} C_VEL
LIN {X 0,Y 580.695,Z 306.817,A -85,B 0,C 180,E1 -1728.981,E2 -1728.981} C_VEL
LIN {X 0,Y 580.839,Z 294.25,A -85,B 0,C 180,E1 -1729.642,E2 -1729.642} C_VEL
LIN {X 0,Y 580.999,Z 281.524,A -85,B 0,C 180,E1 -1730.166,E2 -1730.166} C_VEL
LIN {X 0,Y 581.032,Z 268.107,A -85,B 0,C 180,E1 -1730.581,E2 -1730.581} C_VEL
LIN {X 0,Y 581.117,Z 253.51,A -85,B 0,C 180,E1 -1730.879,E2 -1730.879} C_VEL
LIN {X 0,Y 581.258,Z 123.779,A -85,B 0,C 180,E1 -1732.515,E2 -1732.515} C_VEL
LIN {X 0,Y 580.493,Z 119.541,A -85,B 0,C 180,E1 -1732.606,E2 -1732.606} C_VEL
LIN {X 0,Y 580.642,Z 100.499,A -85,B 0,C 180,E1 -1735.448,E2 -1735.448} C_VEL
LIN {X 0,Y 580.68,Z 89.081,A -85,B 0,C 180,E1 -1737.187,E2 -1737.187} C_VEL
LIN {X 0,Y 580.226,Z 86.337,A -85,B 0,C 180,E1 -1737.653,E2 -1737.653} C_VEL
LIN {X 0,Y 580.268,Z 86.329,A -85,B 0,C 180,E1 -1740.577,E2 -1740.577} C_VEL
LIN {X 0,Y 580.267,Z 86.325,A -85,B 0,C 180,E1 -1743.31,E2 -1743.31} C_VEL
LIN {X 0,Y 580.219,Z 86.337,A -85,B 0,C 180,E1 -1745.752,E2 -1745.752} C_VEL
LIN {X 0,Y 580.266,Z 86.33,A -85,B 0,C 180,E1 -1748.148,E2 -1748.148} C_VEL
LIN {X 0,Y 580.24,Z 86.328,A -85,B 0,C 180,E1 -1750.848,E2 -1750.848} C_VEL
LIN {X 0,Y 580.225,Z 86.339,A -85,B 0,C 180,E1 -1753.663,E2 -1753.663} C_VEL
LIN {X 0,Y 580.235,Z 86.328,A -85,B 0,C 180,E1 -1756.614,E2 -1756.614} C_VEL
LIN {X 0,Y 580.271,Z 86.329,A -85,B 0,C 180,E1 -1759.154,E2 -1759.154} C_VEL
LIN {X 0,Y 580.275,Z 86.325,A -85,B 0,C 180,E1 -1761.929,E2 -1761.929} C_VEL
LIN {X 0,Y 580.231,Z 86.329,A -85,B 0,C 180,E1 -1764.451,E2 -1764.451} C_VEL
LIN {X 0,Y 580.284,Z 86.329,A -85,B 0,C 180,E1 -1766.974,E2 -1766.974} C_VEL
LIN {X 0,Y 580.27,Z 86.327,A -85,B 0,C 180,E1 -1769.423,E2 -1769.423} C_VEL
LIN {X 0,Y 580.248,Z 86.327,A -85,B 0,C 180,E1 -1772.151,E2 -1772.151} C_VEL
LIN {X 0,Y 580.274,Z 86.333,A -85,B 0,C 180,E1 -1774.919,E2 -1774.919} C_VEL
LIN {X 0,Y 580.251,Z 86.326,A -85,B 0,C 180,E1 -1777.946,E2 -1777.946} C_VEL
LIN {X 0,Y 580.298,Z 86.326,A -85,B 0,C 180,E1 -1780.849,E2 -1780.849} C_VEL
LIN {X 0,Y 580.257,Z 86.326,A -85,B 0,C 180,E1 -1783.825,E2 -1783.825} C_VEL
LIN {X 0,Y 580.257,Z 86.331,A -85,B 0,C 180,E1 -1786.695,E2 -1786.695} C_VEL
LIN {X 0,Y 580.307,Z 86.322,A -85,B 0,C 180,E1 -1788.827,E2 -1788.827} C_VEL
LIN {X 0,Y 580.306,Z 86.319,A -85,B 0,C 180,E1 -1791.643,E2 -1791.643} C_VEL
LIN {X 0,Y 580.323,Z 86.322,A -85,B 0,C 180,E1 -1794.44,E2 -1794.44} C_VEL
LIN {X 0,Y 580.323,Z 86.317,A -85,B 0,C 180,E1 -1797.223,E2 -1797.223} C_VEL
LIN {X 0,Y 580.354,Z 86.321,A -85,B 0,C 180,E1 -1800,E2 -1800} C_VEL
LIN {X 0,Y 580.334,Z 86.316,A -85,B 0,C 180,E1 -1802.776,E2 -1802.776} C_VEL
LIN {X 0,Y 580.313,Z 86.325,A -85,B 0,C 180,E1 -1805.56,E2 -1805.56} C_VEL
LIN {X 0,Y 580.326,Z 86.318,A -85,B 0,C 180,E1 -1808.356,E2 -1808.356} C_VEL
LIN {X 0,Y 580.302,Z 86.324,A -85,B 0,C 180,E1 -1811.191,E2 -1811.191} C_VEL
LIN {X 0,Y 580.315,Z 86.32,A -85,B 0,C 180,E1 -1814.017,E2 -1814.017} C_VEL
LIN {X 0,Y 580.314,Z 86.32,A -85,B 0,C 180,E1 -1816.914,E2 -1816.914} C_VEL
LIN {X 0,Y 580.287,Z 86.322,A -85,B 0,C 180,E1 -1819.823,E2 -1819.823} C_VEL
LIN {X 0,Y 580.267,Z 86.324,A -85,B 0,C 180,E1 -1822.053,E2 -1822.053} C_VEL
LIN {X 0,Y 580.308,Z 86.328,A -85,B 0,C 180,E1 -1825.08,E2 -1825.08} C_VEL
LIN {X 0,Y 580.298,Z 86.321,A -85,B 0,C 180,E1 -1828.186,E2 -1828.186} C_VEL
LIN {X 0,Y 580.293,Z 86.329,A -85,B 0,C 180,E1 -1830.696,E2 -1830.696} C_VEL
LIN {X 0,Y 580.305,Z 86.321,A -85,B 0,C 180,E1 -1833.316,E2 -1833.316} C_VEL
LIN {X 0,Y 580.25,Z 86.326,A -85,B 0,C 180,E1 -1835.757,E2 -1835.757} C_VEL
LIN {X 0,Y 580.287,Z 86.326,A -85,B 0,C 180,E1 -1838.146,E2 -1838.146} C_VEL
LIN {X 0,Y 580.299,Z 86.324,A -85,B 0,C 180,E1 -1840.843,E2 -1840.843} C_VEL
LIN {X 0,Y 580.281,Z 86.323,A -85,B 0,C 180,E1 -1843.658,E2 -1843.658} C_VEL
LIN {X 0,Y 580.274,Z 86.327,A -85,B 0,C 180,E1 -1846.61,E2 -1846.61} C_VEL
LIN {X 0,Y 580.3,Z 86.32,A -85,B 0,C 180,E1 -1849.157,E2 -1849.157} C_VEL
LIN {X 0,Y 580.292,Z 86.329,A -85,B 0,C 180,E1 -1851.927,E2 -1851.927} C_VEL
LIN {X 0,Y 580.253,Z 86.328,A -85,B 0,C 180,E1 -1854.453,E2 -1854.453} C_VEL
LIN {X 0,Y 580.291,Z 86.32,A -85,B 0,C 180,E1 -1856.975,E2 -1856.975} C_VEL
LIN {X 0,Y 580.297,Z 86.325,A -85,B 0,C 180,E1 -1859.425,E2 -1859.425} C_VEL
LIN {X 0,Y 580.3,Z 86.324,A -85,B 0,C 180,E1 -1862.141,E2 -1862.141} C_VEL
LIN {X 0,Y 580.323,Z 86.325,A -85,B 0,C 180,E1 -1865.27,E2 -1865.27} C_VEL
LIN {X 0,Y 580.328,Z 86.438,A -85,B 0,C 180,E1 -1865.875,E2 -1865.875} C_VEL
LIN {X 0,Y 581.092,Z 90.674,A -85,B 0,C 180,E1 -1866.477,E2 -1866.477} C_VEL
LIN {X 0,Y 580.907,Z 111.812,A -85,B 0,C 180,E1 -1869.275,E2 -1869.275} C_VEL
LIN {X 0,Y 580.713,Z 132.751,A -85,B 0,C 180,E1 -1872.024,E2 -1872.024} C_VEL
LIN {X 0,Y 580.58,Z 143.697,A -85,B 0,C 180,E1 -1873.444,E2 -1873.444} C_VEL
LIN {X 0,Y 581.405,Z 149.397,A -85,B 0,C 180,E1 -1873.542,E2 -1873.542} C_VEL
LIN {X 0,Y 581.119,Z 281.88,A -85,B 0,C 180,E1 -1875.22,E2 -1875.22} C_VEL
LIN {X 0,Y 581.043,Z 296.459,A -85,B 0,C 180,E1 -1875.556,E2 -1875.556} C_VEL
LIN {X 0,Y 580.895,Z 310.836,A -85,B 0,C 180,E1 -1876.042,E2 -1876.042} C_VEL
LIN {X 0,Y 580.787,Z 323.641,A -85,B 0,C 180,E1 -1876.619,E2 -1876.619} C_VEL
LIN {X 0,Y 580.655,Z 336.1,A -85,B 0,C 180,E1 -1877.327,E2 -1877.327} C_VEL
LIN {X 0,Y 580.525,Z 348.642,A -85,B 0,C 180,E1 -1878.212,E2 -1878.212} C_VEL
LIN {X 0,Y 580.441,Z 359.891,A -85,B 0,C 180,E1 -1879.189,E2 -1879.189} C_VEL
LIN {X 0,Y 580.276,Z 369.851,A -85,B 0,C 180,E1 -1880.238,E2 -1880.238} C_VEL
LIN {X 0,Y 580.241,Z 378.172,A -85,B 0,C 180,E1 -1881.292,E2 -1881.292} C_VEL
LIN {X 0,Y 580.166,Z 386.126,A -85,B 0,C 180,E1 -1882.517,E2 -1882.517} C_VEL
LIN {X 0,Y 580.103,Z 392.527,A -85,B 0,C 180,E1 -1883.74,E2 -1883.74} C_VEL
LIN {X 0,Y 580.077,Z 396.961,A -85,B 0,C 180,E1 -1884.786,E2 -1884.786} C_VEL
LIN {X 0,Y 580.103,Z 400.443,A -85,B 0,C 180,E1 -1885.831,E2 -1885.831} C_VEL
LIN {X 0,Y 580.04,Z 403.831,A -85,B 0,C 180,E1 -1887.222,E2 -1887.222} C_VEL
LIN {X 0,Y 580.042,Z 405.832,A -85,B 0,C 180,E1 -1888.611,E2 -1888.611} C_VEL
LIN {X 0,Y 580.036,Z 406.5,A -85,B 0,C 180,E1 -1890,E2 -1890} C_VEL
LIN {X 0,Y 580.042,Z 405.833,A -85,B 0,C 180,E1 -1891.388,E2 -1891.388} C_VEL
LIN {X 0,Y 580.04,Z 403.834,A -85,B 0,C 180,E1 -1892.778,E2 -1892.778} C_VEL
LIN {X 0,Y 580.103,Z 400.445,A -85,B 0,C 180,E1 -1894.168,E2 -1894.168} C_VEL
LIN {X 0,Y 580.128,Z 395.568,A -85,B 0,C 180,E1 -1895.562,E2 -1895.562} C_VEL
LIN {X 0,Y 580.141,Z 389.054,A -85,B 0,C 180,E1 -1896.958,E2 -1896.958} C_VEL
LIN {X 0,Y 580.192,Z 381.802,A -85,B 0,C 180,E1 -1898.183,E2 -1898.183} C_VEL
LIN {X 0,Y 580.283,Z 372.823,A -85,B 0,C 180,E1 -1899.41,E2 -1899.41} C_VEL
LIN {X 0,Y 580.356,Z 363.393,A -85,B 0,C 180,E1 -1900.466,E2 -1900.466} C_VEL
LIN {X 0,Y 580.477,Z 353.323,A -85,B 0,C 180,E1 -1901.404,E2 -1901.404} C_VEL
LIN {X 0,Y 580.617,Z 341.437,A -85,B 0,C 180,E1 -1902.318,E2 -1902.318} C_VEL
LIN {X 0,Y 580.723,Z 328.646,A -85,B 0,C 180,E1 -1903.115,E2 -1903.115} C_VEL
LIN {X 0,Y 580.849,Z 316.156,A -85,B 0,C 180,E1 -1903.736,E2 -1903.736} C_VEL
LIN {X 0,Y 581.019,Z 303.248,A -85,B 0,C 180,E1 -1904.233,E2 -1904.233} C_VEL
LIN {X 0,Y 581.082,Z 289.197,A -85,B 0,C 180,E1 -1904.63,E2 -1904.63} C_VEL
LIN {X 0,Y 581.16,Z 274.612,A -85,B 0,C 180,E1 -1904.891,E2 -1904.891} C_VEL
LIN {X 0,Y 581.343,Z 147.852,A -85,B 0,C 180,E1 -1906.479,E2 -1906.479} C_VEL
LIN {X 0,Y 580.571,Z 143.568,A -85,B 0,C 180,E1 -1906.573,E2 -1906.573} C_VEL
LIN {X 0,Y 580.727,Z 124.38,A -85,B 0,C 180,E1 -1909.072,E2 -1909.072} C_VEL
LIN {X 0,Y 580.913,Z 104.774,A -85,B 0,C 180,E1 -1911.653,E2 -1911.653} C_VEL
LIN {X 0,Y 581.092,Z 90.679,A -85,B 0,C 180,E1 -1913.523,E2 -1913.523} C_VEL
LIN {X 0,Y 580.309,Z 86.326,A -85,B 0,C 180,E1 -1914.173,E2 -1914.173} C_VEL
LIN {X 0,Y 580.278,Z 86.33,A -85,B 0,C 180,E1 -1916.623,E2 -1916.623} C_VEL
LIN {X 0,Y 580.302,Z 86.32,A -85,B 0,C 180,E1 -1919.309,E2 -1919.309} C_VEL
LIN {X 0,Y 580.299,Z 86.33,A -85,B 0,C 180,E1 -1922.2,E2 -1922.2} C_VEL
LIN {X 0,Y 580.29,Z 86.323,A -85,B 0,C 180,E1 -1924.696,E2 -1924.696} C_VEL
LIN {X 0,Y 580.299,Z 86.32,A -85,B 0,C 180,E1 -1927.268,E2 -1927.268} C_VEL
LIN {X 0,Y 580.297,Z 86.325,A -85,B 0,C 180,E1 -1930.271,E2 -1930.271} C_VEL
LIN {X 0,Y 580.276,Z 86.323,A -85,B 0,C 180,E1 -1932.706,E2 -1932.706} C_VEL
LIN {X 0,Y 580.274,Z 86.33,A -85,B 0,C 180,E1 -1935.608,E2 -1935.608} C_VEL
LIN {X 0,Y 580.314,Z 86.32,A -85,B 0,C 180,E1 -1938.234,E2 -1938.234} C_VEL
LIN {X 0,Y 580.277,Z 86.324,A -85,B 0,C 180,E1 -1940.965,E2 -1940.965} C_VEL
LIN {X 0,Y 580.268,Z 86.332,A -85,B 0,C 180,E1 -1943.596,E2 -1943.596} C_VEL
LIN {X 0,Y 580.317,Z 86.318,A -85,B 0,C 180,E1 -1946.145,E2 -1946.145} C_VEL
LIN {X 0,Y 580.28,Z 86.323,A -85,B 0,C 180,E1 -1948.615,E2 -1948.615} C_VEL
LIN {X 0,Y 580.292,Z 86.327,A -85,B 0,C 180,E1 -1951.024,E2 -1951.024} C_VEL
LIN {X 0,Y 580.292,Z 86.324,A -85,B 0,C 180,E1 -1953.666,E2 -1953.666} C_VEL
LIN {X 0,Y 580.3,Z 86.322,A -85,B 0,C 180,E1 -1955.684,E2 -1955.684} C_VEL
LIN {X 0,Y 580.269,Z 86.324,A -85,B 0,C 180,E1 -1957.947,E2 -1957.947} C_VEL
LIN {X 0,Y 580.296,Z 86.33,A -85,B 0,C 180,E1 -1960.913,E2 -1960.913} C_VEL
LIN {X 0,Y 580.27,Z 86.323,A -85,B 0,C 180,E1 -1963.825,E2 -1963.825} C_VEL
LIN {X 0,Y 580.327,Z 86.317,A -85,B 0,C 180,E1 -1965.983,E2 -1965.983} C_VEL
LIN {X 0,Y 580.304,Z 86.327,A -85,B 0,C 180,E1 -1968.827,E2 -1968.827} C_VEL
LIN {X 0,Y 580.327,Z 86.316,A -85,B 0,C 180,E1 -1971.644,E2 -1971.644} C_VEL
LIN {X 0,Y 580.319,Z 86.327,A -85,B 0,C 180,E1 -1974.44,E2 -1974.44} C_VEL
LIN {X 0,Y 580.338,Z 86.315,A -85,B 0,C 180,E1 -1977.224,E2 -1977.224} C_VEL
LIN {X 0,Y 580.352,Z 86.318,A -85,B 0,C 180,E1 -1980,E2 -1980} C_VEL
LIN {X 0,Y 580.333,Z 86.318,A -85,B 0,C 180,E1 -1982.777,E2 -1982.777} C_VEL
LIN {X 0,Y 580.323,Z 86.319,A -85,B 0,C 180,E1 -1985.56,E2 -1985.56} C_VEL
LIN {X 0,Y 580.326,Z 86.321,A -85,B 0,C 180,E1 -1988.356,E2 -1988.356} C_VEL
LIN {X 0,Y 580.3,Z 86.32,A -85,B 0,C 180,E1 -1991.191,E2 -1991.191} C_VEL
LIN {X 0,Y 580.327,Z 86.323,A -85,B 0,C 180,E1 -1994.017,E2 -1994.017} C_VEL
LIN {X 0,Y 580.312,Z 86.319,A -85,B 0,C 180,E1 -1996.914,E2 -1996.914} C_VEL
LIN {X 0,Y 580.301,Z 86.327,A -85,B 0,C 180,E1 -1999.823,E2 -1999.823} C_VEL
LIN {X 0,Y 580.282,Z 86.327,A -85,B 0,C 180,E1 -2001.318,E2 -2001.318} C_VEL
LIN {X 0,Y 579.582,Z 86.414,A -85,B 0,C 180,E1 -2001.897,E2 -2001.897} C_VEL
LIN {X 0,Y 576.703,Z 86.769,A -85,B 0,C 180,E1 -2002.837,E2 -2002.837} C_VEL
LIN {X 0,Y 574.309,Z 87.075,A -85,B 0,C 180,E1 -2003.593,E2 -2003.593} C_VEL
LIN {X 0,Y 573.312,Z 87.192,A -85,B 0,C 180,E1 -2004.177,E2 -2004.177} C_VEL
LIN {X 0,Y 573.246,Z 87.199,A -85,B 0,C 180,E1 -2004.375,E2 -2004.375} C_VEL
LIN {X 0,Y 573.25,Z 87.201,A -85,B 0,C 180,E1 -2006.976,E2 -2006.976} C_VEL
LIN {X 0,Y 573.24,Z 87.207,A -85,B 0,C 180,E1 -2009.487,E2 -2009.487} C_VEL
LIN {X 0,Y 573.252,Z 87.2,A -85,B 0,C 180,E1 -2012.645,E2 -2012.645} C_VEL
LIN {X 0,Y 573.206,Z 87.213,A -85,B 0,C 180,E1 -2015.188,E2 -2015.188} C_VEL
LIN {X 0,Y 573.233,Z 87.201,A -85,B 0,C 180,E1 -2017.808,E2 -2017.808} C_VEL
LIN {X 0,Y 573.245,Z 87.202,A -85,B 0,C 180,E1 -2020.525,E2 -2020.525} C_VEL
LIN {X 0,Y 573.232,Z 87.203,A -85,B 0,C 180,E1 -2023.36,E2 -2023.36} C_VEL
LIN {X 0,Y 573.237,Z 87.203,A -85,B 0,C 180,E1 -2026.332,E2 -2026.332} C_VEL
LIN {X 0,Y 573.226,Z 87.208,A -85,B 0,C 180,E1 -2028.543,E2 -2028.543} C_VEL
LIN {X 0,Y 573.238,Z 87.201,A -85,B 0,C 180,E1 -2031.298,E2 -2031.298} C_VEL
LIN {X 0,Y 573.194,Z 87.208,A -85,B 0,C 180,E1 -2034.022,E2 -2034.022} C_VEL
LIN {X 0,Y 573.272,Z 87.204,A -85,B 0,C 180,E1 -2036.518,E2 -2036.518} C_VEL
LIN {X 0,Y 573.228,Z 87.201,A -85,B 0,C 180,E1 -2039.119,E2 -2039.119} C_VEL
LIN {X 0,Y 573.225,Z 87.201,A -85,B 0,C 180,E1 -2041.435,E2 -2041.435} C_VEL
LIN {X 0,Y 573.242,Z 87.202,A -85,B 0,C 180,E1 -2044.59,E2 -2044.59} C_VEL
LIN {X 0,Y 573.233,Z 87.204,A -85,B 0,C 180,E1 -2047.662,E2 -2047.662} C_VEL
LIN {X 0,Y 573.269,Z 87.198,A -85,B 0,C 180,E1 -2050.67,E2 -2050.67} C_VEL
LIN {X 0,Y 573.242,Z 87.208,A -85,B 0,C 180,E1 -2053.622,E2 -2053.622} C_VEL
LIN {X 0,Y 573.244,Z 87.227,A -85,B 0,C 180,E1 -2054.307,E2 -2054.307} C_VEL
LIN {X 0,Y 573.838,Z 90.966,A -85,B 0,C 180,E1 -2054.915,E2 -2054.915} C_VEL
LIN {X 0,Y 573.585,Z 109.746,A -85,B 0,C 180,E1 -2057.798,E2 -2057.798} C_VEL
LIN {X 0,Y 573.52,Z 119.567,A -85,B 0,C 180,E1 -2059.28,E2 -2059.28} C_VEL
LIN {X 0,Y 574.555,Z 126.008,A -85,B 0,C 180,E1 -2059.406,E2 -2059.406} C_VEL
LIN {X 0,Y 574.255,Z 255.978,A -85,B 0,C 180,E1 -2061.067,E2 -2061.067} C_VEL
LIN {X 0,Y 574.174,Z 270.581,A -85,B 0,C 180,E1 -2061.399,E2 -2061.399} C_VEL
LIN {X 0,Y 574.057,Z 284.459,A -85,B 0,C 180,E1 -2061.862,E2 -2061.862} C_VEL
LIN {X 0,Y 573.921,Z 297.372,A -85,B 0,C 180,E1 -2062.436,E2 -2062.436} C_VEL
LIN {X 0,Y 573.718,Z 310.421,A -85,B 0,C 180,E1 -2063.174,E2 -2063.174} C_VEL
LIN {X 0,Y 573.595,Z 322.476,A -85,B 0,C 180,E1 -2064.022,E2 -2064.022} C_VEL
LIN {X 0,Y 573.398,Z 332.802,A -85,B 0,C 180,E1 -2064.902,E2 -2064.902} C_VEL
LIN {X 0,Y 573.282,Z 343.094,A -85,B 0,C 180,E1 -2065.958,E2 -2065.958} C_VEL
LIN {X 0,Y 573.183,Z 351.623,A -85,B 0,C 180,E1 -2067.013,E2 -2067.013} C_VEL
LIN {X 0,Y 573.167,Z 359.828,A -85,B 0,C 180,E1 -2068.243,E2 -2068.243} C_VEL
LIN {X 0,Y 573.024,Z 365.574,A -85,B 0,C 180,E1 -2069.297,E2 -2069.297} C_VEL
LIN {X 0,Y 572.983,Z 371.727,A -85,B 0,C 180,E1 -2070.703,E2 -2070.703} C_VEL
LIN {X 0,Y 572.941,Z 376.257,A -85,B 0,C 180,E1 -2072.109,E2 -2072.109} C_VEL
LIN {X 0,Y 573.003,Z 379.338,A -85,B 0,C 180,E1 -2073.516,E2 -2073.516} C_VEL
LIN {X 0,Y 572.934,Z 381.056,A -85,B 0,C 180,E1 -2074.926,E2 -2074.926} C_VEL
LIN {X 0,Y 572.975,Z 381.441,A -85,B 0,C 180,E1 -2076.338,E2 -2076.338} C_VEL
LIN {X 0,Y 572.976,Z 380.494,A -85,B 0,C 180,E1 -2077.754,E2 -2077.754} C_VEL
LIN {X 0,Y 572.93,Z 378.179,A -85,B 0,C 180,E1 -2079.176,E2 -2079.176} C_VEL
LIN {X 0,Y 573.021,Z 374.43,A -85,B 0,C 180,E1 -2080.601,E2 -2080.601} C_VEL
LIN {X 0,Y 573.021,Z 370.57,A -85,B 0,C 180,E1 -2081.676,E2 -2081.676} C_VEL
LIN {X 0,Y 573.04,Z 365.772,A -85,B 0,C 180,E1 -2082.754,E2 -2082.754} C_VEL
LIN {X 0,Y 573.118,Z 358.776,A -85,B 0,C 180,E1 -2084.016,E2 -2084.016} C_VEL
LIN {X 0,Y 573.198,Z 350.041,A -85,B 0,C 180,E1 -2085.285,E2 -2085.285} C_VEL
LIN {X 0,Y 573.348,Z 340.864,A -85,B 0,C 180,E1 -2086.375,E2 -2086.375} C_VEL
LIN {X 0,Y 573.418,Z 331.68,A -85,B 0,C 180,E1 -2087.291,E2 -2087.291} C_VEL
LIN {X 0,Y 573.597,Z 320.666,A -85,B 0,C 180,E1 -2088.206,E2 -2088.206} C_VEL
LIN {X 0,Y 573.754,Z 308.538,A -85,B 0,C 180,E1 -2089.034,E2 -2089.034} C_VEL
LIN {X 0,Y 573.901,Z 295.6,A -85,B 0,C 180,E1 -2089.745,E2 -2089.745} C_VEL
LIN {X 0,Y 574.11,Z 281.922,A -85,B 0,C 180,E1 -2090.326,E2 -2090.326} C_VEL
LIN {X 0,Y 574.191,Z 267.738,A -85,B 0,C 180,E1 -2090.767,E2 -2090.767} C_VEL
LIN {X 0,Y 574.281,Z 253.113,A -85,B 0,C 180,E1 -2091.066,E2 -2091.066} C_VEL
LIN {X 0,Y 574.508,Z 124.878,A -85,B 0,C 180,E1 -2092.7,E2 -2092.7} C_VEL
LIN {X 0,Y 573.529,Z 119.465,A -85,B 0,C 180,E1 -2092.825,E2 -2092.825} C_VEL
LIN {X 0,Y 573.709,Z 100.03,A -85,B 0,C 180,E1 -2095.778,E2 -2095.778} C_VEL
LIN {X 0,Y 573.8,Z 91.174,A -85,B 0,C 180,E1 -2097.145,E2 -2097.145} C_VEL
LIN {X 0,Y 573.185,Z 87.215,A -85,B 0,C 180,E1 -2097.814,E2 -2097.814} C_VEL
LIN {X 0,Y 573.219,Z 87.212,A -85,B 0,C 180,E1 -2100.178,E2 -2100.178} C_VEL
LIN {X 0,Y 573.22,Z 87.204,A -85,B 0,C 180,E1 -2102.647,E2 -2102.647} C_VEL
LIN {X 0,Y 573.181,Z 87.208,A -85,B 0,C 180,E1 -2105.19,E2 -2105.19} C_VEL
LIN {X 0,Y 573.211,Z 87.212,A -85,B 0,C 180,E1 -2107.81,E2 -2107.81} C_VEL
LIN {X 0,Y 573.203,Z 87.205,A -85,B 0,C 180,E1 -2110.529,E2 -2110.529} C_VEL
LIN {X 0,Y 573.189,Z 87.211,A -85,B 0,C 180,E1 -2113.364,E2 -2113.364} C_VEL
LIN {X 0,Y 573.205,Z 87.204,A -85,B 0,C 180,E1 -2116.335,E2 -2116.335} C_VEL
LIN {X 0,Y 573.197,Z 87.205,A -85,B 0,C 180,E1 -2118.54,E2 -2118.54} C_VEL
LIN {X 0,Y 573.229,Z 87.207,A -85,B 0,C 180,E1 -2121.297,E2 -2121.297} C_VEL
LIN {X 0,Y 573.188,Z 87.206,A -85,B 0,C 180,E1 -2124.022,E2 -2124.022} C_VEL
LIN {X 0,Y 573.227,Z 87.202,A -85,B 0,C 180,E1 -2126.515,E2 -2126.515} C_VEL
LIN {X 0,Y 573.215,Z 87.211,A -85,B 0,C 180,E1 -2129.12,E2 -2129.12} C_VEL
LIN {X 0,Y 573.204,Z 87.207,A -85,B 0,C 180,E1 -2131.433,E2 -2131.433} C_VEL
LIN {X 0,Y 573.223,Z 87.206,A -85,B 0,C 180,E1 -2134.588,E2 -2134.588} C_VEL
LIN {X 0,Y 573.219,Z 87.201,A -85,B 0,C 180,E1 -2137.661,E2 -2137.661} C_VEL
LIN {X 0,Y 573.235,Z 87.201,A -85,B 0,C 180,E1 -2139.923,E2 -2139.923} C_VEL
LIN {X 0,Y 573.237,Z 87.203,A -85,B 0,C 180,E1 -2142.998,E2 -2142.998} C_VEL
LIN {X 0,Y 573.234,Z 87.201,A -85,B 0,C 180,E1 -2145.806,E2 -2145.806} C_VEL
LIN {X 0,Y 573.264,Z 87.2,A -85,B 0,C 180,E1 -2148.745,E2 -2148.745} C_VEL
LIN {X 0,Y 573.251,Z 87.197,A -85,B 0,C 180,E1 -2151.54,E2 -2151.54} C_VEL
LIN {X 0,Y 573.289,Z 87.199,A -85,B 0,C 180,E1 -2154.372,E2 -2154.372} C_VEL
LIN {X 0,Y 573.311,Z 87.198,A -85,B 0,C 180,E1 -2157.892,E2 -2157.892} C_VEL
LIN {X 0,Y 573.327,Z 87.188,A -85,B 0,C 180,E1 -2160.702,E2 -2160.702} C_VEL
LIN {X 0,Y 573.3,Z 87.192,A -85,B 0,C 180,E1 -2162.811,E2 -2162.811} C_VEL
LIN {X 0,Y 573.28,Z 87.202,A -85,B 0,C 180,E1 -2165.628,E2 -2165.628} C_VEL
LIN {X 0,Y 573.282,Z 87.195,A -85,B 0,C 180,E1 -2168.459,E2 -2168.459} C_VEL
LIN {X 0,Y 573.273,Z 87.201,A -85,B 0,C 180,E1 -2171.312,E2 -2171.312} C_VEL
LIN {X 0,Y 573.269,Z 87.196,A -85,B 0,C 180,E1 -2174.419,E2 -2174.419} C_VEL
LIN {X 0,Y 573.259,Z 87.202,A -85,B 0,C 180,E1 -2177.111,E2 -2177.111} C_VEL
LIN {X 0,Y 573.241,Z 87.199,A -85,B 0,C 180,E1 -2180.077,E2 -2180.077} C_VEL
LIN {X 0,Y 573.232,Z 87.2,A -85,B 0,C 180,E1 -2182.338,E2 -2182.338} C_VEL
LIN {X 0,Y 573.256,Z 87.201,A -85,B 0,C 180,E1 -2185.41,E2 -2185.41} C_VEL
LIN {X 0,Y 573.251,Z 87.198,A -85,B 0,C 180,E1 -2188.029,E2 -2188.029} C_VEL
LIN {X 0,Y 573.239,Z 87.208,A -85,B 0,C 180,E1 -2190.884,E2 -2190.884} C_VEL
LIN {X 0,Y 573.263,Z 87.197,A -85,B 0,C 180,E1 -2193.524,E2 -2193.524} C_VEL
LIN {X 0,Y 573.216,Z 87.204,A -85,B 0,C 180,E1 -2196.051,E2 -2196.051} C_VEL
LIN {X 0,Y 573.241,Z 87.204,A -85,B 0,C 180,E1 -2198.702,E2 -2198.702} C_VEL
LIN {X 0,Y 573.245,Z 87.199,A -85,B 0,C 180,E1 -2201.594,E2 -2201.594} C_VEL
LIN {X 0,Y 573.234,Z 87.208,A -85,B 0,C 180,E1 -2204.334,E2 -2204.334} C_VEL
LIN {X 0,Y 573.241,Z 87.2,A -85,B 0,C 180,E1 -2207.359,E2 -2207.359} C_VEL
LIN {X 0,Y 573.249,Z 87.203,A -85,B 0,C 180,E1 -2210.393,E2 -2210.393} C_VEL
LIN {X 0,Y 573.254,Z 87.198,A -85,B 0,C 180,E1 -2213.078,E2 -2213.078} C_VEL
LIN {X 0,Y 573.269,Z 87.202,A -85,B 0,C 180,E1 -2215.671,E2 -2215.671} C_VEL
LIN {X 0,Y 573.242,Z 87.203,A -85,B 0,C 180,E1 -2218.185,E2 -2218.185} C_VEL
LIN {X 0,Y 573.265,Z 87.197,A -85,B 0,C 180,E1 -2220.634,E2 -2220.634} C_VEL
LIN {X 0,Y 573.253,Z 87.201,A -85,B 0,C 180,E1 -2223.024,E2 -2223.024} C_VEL
LIN {X 0,Y 573.293,Z 87.359,A -85,B 0,C 180,E1 -2225.704,E2 -2225.704} C_VEL
LIN {X 0,Y 574.187,Z 92.676,A -85,B 0,C 180,E1 -2226.468,E2 -2226.468} C_VEL
LIN {X 0,Y 573.958,Z 113.075,A -85,B 0,C 180,E1 -2229.2,E2 -2229.2} C_VEL
LIN {X 0,Y 573.743,Z 134.146,A -85,B 0,C 180,E1 -2231.983,E2 -2231.983} C_VEL
LIN {X 0,Y 573.632,Z 143.709,A -85,B 0,C 180,E1 -2233.24,E2 -2233.24} C_VEL
LIN {X 0,Y 574.593,Z 149.497,A -85,B 0,C 180,E1 -2233.342,E2 -2233.342} C_VEL
LIN {X 0,Y 574.25,Z 281.88,A -85,B 0,C 180,E1 -2235.039,E2 -2235.039} C_VEL
LIN {X 0,Y 574.145,Z 296.458,A -85,B 0,C 180,E1 -2235.379,E2 -2235.379} C_VEL
LIN {X 0,Y 573.989,Z 310.834,A -85,B 0,C 180,E1 -2235.87,E2 -2235.87} C_VEL
LIN {X 0,Y 573.873,Z 323.639,A -85,B 0,C 180,E1 -2236.454,E2 -2236.454} C_VEL
LIN {X 0,Y 573.716,Z 336.101,A -85,B 0,C 180,E1 -2237.172,E2 -2237.172} C_VEL
LIN {X 0,Y 573.532,Z 348.644,A -85,B 0,C 180,E1 -2238.066,E2 -2238.066} C_VEL
LIN {X 0,Y 573.437,Z 360.141,A -85,B 0,C 180,E1 -2239.08,E2 -2239.08} C_VEL
LIN {X 0,Y 573.24,Z 369.851,A -85,B 0,C 180,E1 -2240.117,E2 -2240.117} C_VEL
LIN {X 0,Y 573.202,Z 378.173,A -85,B 0,C 180,E1 -2241.184,E2 -2241.184} C_VEL
LIN {X 0,Y 573.11,Z 386.127,A -85,B 0,C 180,E1 -2242.425,E2 -2242.425} C_VEL
LIN {X 0,Y 573.021,Z 392.527,A -85,B 0,C 180,E1 -2243.662,E2 -2243.662} C_VEL
LIN {X 0,Y 573,Z 396.961,A -85,B 0,C 180,E1 -2244.722,E2 -2244.722} C_VEL
LIN {X 0,Y 573.029,Z 400.443,A -85,B 0,C 180,E1 -2245.78,E2 -2245.78} C_VEL
LIN {X 0,Y 572.955,Z 403.832,A -85,B 0,C 180,E1 -2247.188,E2 -2247.188} C_VEL
LIN {X 0,Y 572.941,Z 405.833,A -85,B 0,C 180,E1 -2248.594,E2 -2248.594} C_VEL
LIN {X 0,Y 572.936,Z 406.5,A -85,B 0,C 180,E1 -2250,E2 -2250} C_VEL
LIN {X 0,Y 572.941,Z 405.834,A -85,B 0,C 180,E1 -2251.406,E2 -2251.406} C_VEL
LIN {X 0,Y 572.955,Z 403.834,A -85,B 0,C 180,E1 -2252.812,E2 -2252.812} C_VEL
LIN {X 0,Y 573.029,Z 400.446,A -85,B 0,C 180,E1 -2254.22,E2 -2254.22} C_VEL
LIN {X 0,Y 573.057,Z 395.568,A -85,B 0,C 180,E1 -2255.63,E2 -2255.63} C_VEL
LIN {X 0,Y 573.065,Z 390.818,A -85,B 0,C 180,E1 -2256.699,E2 -2256.699} C_VEL
LIN {X 0,Y 573.126,Z 384.037,A -85,B 0,C 180,E1 -2257.929,E2 -2257.929} C_VEL
LIN {X 0,Y 573.225,Z 375.559,A -85,B 0,C 180,E1 -2259.171,E2 -2259.171} C_VEL
LIN {X 0,Y 573.304,Z 366.708,A -85,B 0,C 180,E1 -2260.239,E2 -2260.239} C_VEL
LIN {X 0,Y 573.462,Z 355.99,A -85,B 0,C 180,E1 -2261.308,E2 -2261.308} C_VEL
LIN {X 0,Y 573.62,Z 345.14,A -85,B 0,C 180,E1 -2262.201,E2 -2262.201} C_VEL
LIN {X 0,Y 573.76,Z 333.256,A -85,B 0,C 180,E1 -2263.007,E2 -2263.007} C_VEL
LIN {X 0,Y 573.935,Z 320.098,A -85,B 0,C 180,E1 -2263.724,E2 -2263.724} C_VEL
LIN {X 0,Y 574.121,Z 306.835,A -85,B 0,C 180,E1 -2264.283,E2 -2264.283} C_VEL
LIN {X 0,Y 574.2,Z 292.834,A -85,B 0,C 180,E1 -2264.719,E2 -2264.719} C_VEL
LIN {X 0,Y 574.305,Z 279.138,A -85,B 0,C 180,E1 -2265.005,E2 -2265.005} C_VEL
LIN {X 0,Y 574.513,Z 148.747,A -85,B 0,C 180,E1 -2266.669,E2 -2266.669} C_VEL
LIN {X 0,Y 573.61,Z 143.595,A -85,B 0,C 180,E1 -2266.776,E2 -2266.776} C_VEL
LIN {X 0,Y 573.845,Z 123.411,A -85,B 0,C 180,E1 -2269.432,E2 -2269.432} C_VEL
LIN {X 0,Y 574.062,Z 101.81,A -85,B 0,C 180,E1 -2272.304,E2 -2272.304} C_VEL
LIN {X 0,Y 574.148,Z 91.615,A -85,B 0,C 180,E1 -2273.68,E2 -2273.68} C_VEL
LIN {X 0,Y 573.274,Z 87.205,A -85,B 0,C 180,E1 -2274.344,E2 -2274.344} C_VEL
LIN {X 0,Y 573.252,Z 87.201,A -85,B 0,C 180,E1 -2276.976,E2 -2276.976} C_VEL
LIN {X 0,Y 573.247,Z 87.2,A -85,B 0,C 180,E1 -2279.488,E2 -2279.488} C_VEL
LIN {X 0,Y 573.254,Z 87.201,A -85,B 0,C 180,E1 -2282.645,E2 -2282.645} C_VEL
LIN {X 0,Y 573.208,Z 87.203,A -85,B 0,C 180,E1 -2285.188,E2 -2285.188} C_VEL
LIN {X 0,Y 573.237,Z 87.206,A -85,B 0,C 180,E1 -2287.807,E2 -2287.807} C_VEL
LIN {X 0,Y 573.27,Z 87.197,A -85,B 0,C 180,E1 -2290.528,E2 -2290.528} C_VEL
LIN {X 0,Y 573.244,Z 87.206,A -85,B 0,C 180,E1 -2293.669,E2 -2293.669} C_VEL
LIN {X 0,Y 573.247,Z 87.198,A -85,B 0,C 180,E1 -2296.642,E2 -2296.642} C_VEL
LIN {X 0,Y 573.243,Z 87.206,A -85,B 0,C 180,E1 -2299.475,E2 -2299.475} C_VEL
LIN {X 0,Y 573.234,Z 87.201,A -85,B 0,C 180,E1 -2302.192,E2 -2302.192} C_VEL
LIN {X 0,Y 573.236,Z 87.206,A -85,B 0,C 180,E1 -2305.228,E2 -2305.228} C_VEL
LIN {X 0,Y 573.252,Z 87.201,A -85,B 0,C 180,E1 -2307.771,E2 -2307.771} C_VEL
LIN {X 0,Y 573.264,Z 87.197,A -85,B 0,C 180,E1 -2310.634,E2 -2310.634} C_VEL
LIN {X 0,Y 573.237,Z 87.204,A -85,B 0,C 180,E1 -2313.507,E2 -2313.507} C_VEL
LIN {X 0,Y 573.231,Z 87.2,A -85,B 0,C 180,E1 -2316.135,E2 -2316.135} C_VEL
LIN {X 0,Y 573.249,Z 87.205,A -85,B 0,C 180,E1 -2319.174,E2 -2319.174} C_VEL
LIN {X 0,Y 573.22,Z 87.204,A -85,B 0,C 180,E1 -2321.411,E2 -2321.411} C_VEL
LIN {X 0,Y 573.243,Z 87.199,A -85,B 0,C 180,E1 -2323.622,E2 -2323.622} C_VEL
LIN {X 0,Y 573.273,Z 87.195,A -85,B 0,C 180,E1 -2325.807,E2 -2325.807} C_VEL
LIN {X 0,Y 573.262,Z 87.205,A -85,B 0,C 180,E1 -2328.745,E2 -2328.745} C_VEL
LIN {X 0,Y 573.283,Z 87.194,A -85,B 0,C 180,E1 -2331.541,E2 -2331.541} C_VEL
LIN {X 0,Y 573.286,Z 87.201,A -85,B 0,C 180,E1 -2334.372,E2 -2334.372} C_VEL
LIN {X 0,Y 573.308,Z 87.193,A -85,B 0,C 180,E1 -2337.893,E2 -2337.893} C_VEL
LIN {X 0,Y 573.328,Z 87.192,A -85,B 0,C 180,E1 -2340.702,E2 -2340.702} C_VEL
LIN {X 0,Y 573.235,Z 87.201,A -85,B 0,C 180,E1 -2343.515,E2 -2343.515} C_VEL
